(* CODESYS project SPT_Components.library
   Company: Beckhoff Automation LLC
   DefaultNamespace: SPT_Components
   Version: 3.9.2
   Placeholder: SPT Components
   Title: SPT Components

Project tree, tasks and I/O mapping:
  libraries: SPT Base Types, * (Beckhoff Automation LLC); SPT Event Logger, * (Beckhoff Automation LLC); SPT Motion Control, * (Beckhoff Automation LLC); SPT Utilities, * (Beckhoff Automation LLC); Tc2_DataExchange, * (Beckhoff Automation GmbH); Tc2_EtherCAT, * (Beckhoff Automation GmbH); Tc2_MC2, * (Beckhoff Automation GmbH); Tc2_ModbusRTU, * (Beckhoff Automation GmbH); Tc2_Standard, * (Beckhoff Automation GmbH); Tc2_System, * (Beckhoff Automation GmbH); Tc2_Utilities, * (Beckhoff Automation GmbH); Tc3_EventLogger, * (Beckhoff Automation GmbH); Tc3_Module, * (Beckhoff Automation GmbH); Tc3_PackML_V2, * (Beckhoff Automation GmbH)
  Axes/
    DUT/
      data type ST_AxisBase_Command
      data type ST_AxisBase_Config
      data type ST_AxisBase_HMI
      data type ST_AxisBase_Status
    function block FB_Component_BasicAxis [ST]: Disable, Enable, Home, Jog, MoveAbsolute, MoveModulo, MoveRelative, MoveVelocity, ReadParameterSet, Reset, RunExternalSequence, Stop, WriteBoolParameter, WriteParameter, Acceleration, Deceleration, Jerk, Velocity, ActualAcceleration, ActualPosition, ActualPositionModulo, ActualTorque, ActualVelocity, PositionLag, SetAcceleration, SetPosition, SetPositionModulo, SetVelocity, Enabled, InPosition, Stopped, Axis, AxisParameters, ExternalSequence, HomeMethod, InhibitFeedNegative, InhibitFeedPositive, Override, ResetMethod, CreateEvents, HMICommunication, Monitoring, CyclicLogic, Initialize
    function block FB_Component_BasicSlaveAxis [ST]: Disable, Enable, Home, Jog, MoveAbsolute, MoveModulo, MoveRelative, MoveVelocity, ReadParameterSet, Reset, RunExternalSequence, Stop, WriteBoolParameter, WriteParameter, Acceleration, Deceleration, Jerk, Velocity, ActualAcceleration, ActualPosition, ActualPositionModulo, ActualTorque, ActualVelocity, PositionLag, SetAcceleration, SetPosition, SetPositionModulo, SetVelocity, Enabled, InPosition, Stopped, Axis, AxisParameters, ExternalSequence, HomeMethod, InhibitFeedNegative, InhibitFeedPositive, Override, ResetMethod, GearIn, GearOut, InGear, Master1, Master2, Master3, Master4, RatioMaster1, RatioMaster2, RatioMaster3, RatioMaster4, CreateEvents, HMICommunication, Monitoring, CyclicLogic, Initialize
    function block FB_Component_CamSlaveAxis [ST]: Disable, Enable, Home, Jog, MoveAbsolute, MoveModulo, MoveRelative, MoveVelocity, ReadParameterSet, Reset, RunExternalSequence, Stop, WriteBoolParameter, WriteParameter, Acceleration, Deceleration, Jerk, Velocity, ActualAcceleration, ActualPosition, ActualPositionModulo, ActualTorque, ActualVelocity, PositionLag, SetAcceleration, SetPosition, SetPositionModulo, SetVelocity, Enabled, InPosition, Stopped, Axis, AxisParameters, ExternalSequence, HomeMethod, InhibitFeedNegative, InhibitFeedPositive, Override, ResetMethod, CamParameters, ChangeMode, FindSlavePos, FindSyncPos, InSync, Master, RunningTable, StartCouple, StartSync, SyncPos, UpdateTable, WaitingForCommand, CreateEvents, HMICommunication, Monitoring, CyclicLogic, Initialize
  Communications/
    Modbus-RTU/
      function block FB_Component_ModbusRTUMaster [ST]: CreateEvents, CyclicLogic, Initialize, Monitoring, Reset, RegisterAsyncRequest, RegisterSyncRequest, ProcessRead, ProcessWrite
      function block FB_ModbusAsyncQueue [ST]: Clear, Count, Dequeue, Enqueue, NextRequest
      function block FB_ModbusSyncQueue [ST]: Clear, Count, Enqueue, NextRequest
      interface I_ModbusConsumer: ModbusRequestComplete, SlaveID
      interface I_ModbusProvider: RegisterAsyncRequest, RegisterSyncRequest
      global variables Parameters_ModbusRTU
      data type ST_ModbusOperation
      data type ST_ModbusRequest
  GVLs/
    global variables CONSTANTS
  PackML/
    DUT/
      data type ST_EventInfo
      data type ST_PackML_aEventInfo
      data type ST_PackML_aMsgState
    function block FB_Component_PackML_EventHandler [ST]: AdminTag, AlarmArrayHandler, AlarmToStopReason, AllowHMIControl, BlockHMIControl, Busy, ClearStopReason, ConfirmAlarm, CurrentAlarmSeverity, CyclicLogic, Error, ErrorID, EventListener, Execute, GetMsgInfos, InitComplete, Initialize, InSimulation, InternalErrorAck, MoveAlarmToHistory, Name, OnAlarmCleared, OnAlarmConfirmed, OnAlarmRaised, ParentResponseDefinitions, Reset, TimeZone, WarningToStopReason, WriteAlarmTags
  Project Information/
    function F_GetCompany [ST]
    function F_GetTitle [ST]
    function F_GetVersion [ST]
  Sensors/
    DUT/
      data type E_DebounceMode
      data type E_SensorSimulationMode
      data type ST_DigitalSensor_Command
      data type ST_DigitalSensor_Config
      data type ST_DigitalSensor_HMI
      data type ST_DigitalSensor_Status
    function block FB_DigitalSensor [ST]: CyclicLogic, Active, DebounceMode, DebounceTime, Inverted, SimulationInput, SimulationMode, SimulationTimeBase, TimeActive, TimeInactive, HMICommunication, Monitoring, ProcessInput
    interface I_DigitalSensorBase: Active, DebounceMode, DebounceTime, Inverted, SimulationInput, SimulationMode, TimeActive, TimeInactive
  Solenoids/
    DUT/
      data type ST_Cylinder_Command
      data type ST_Cylinder_Config
      data type ST_Cylinder_HMI
      data type ST_Cylinder_Status
    SolenoidBankBase/
      data type E_SolenoidType
      function block FB_SolenoidBankBase [ST]: AddSolenoid, CheckNumber, CreateEvents, CyclicLogic, Initialize, MapIO, Monitoring, Reset
      data type ST_SolenoidBankConfig
    function block FB_DoubleSolenoid [ST]: HardwareInit, HardwareUpdate, RetractOutput
    function block FB_DoubleSolenoidFeedback [ST]: ExtendedInput, Feedback, HardwareInit, RetractedInput
    function block FB_SingleSolenoid [ST]: CreateEvents, HMICommunication, Monitoring, CyclicLogic, Extend, Extended, ExtendOutput, ExtendTime, Retract, Retracted, RetractOutput, RetractTime, Feedback, HardwareInit, HardwareUpdate, Initialize, Reset
    function block FB_SingleSolenoidFeedback [ST]: ExtendedInput, Feedback, HardwareInit, RetractedInput
    interface I_Solenoid: Extend, Extended, ExtendOutput, ExtendTime, Retract, Retracted, RetractOutput, RetractTime
    global variables Parameters_Cylinder
  Version/
    global variables Global_Version
  00000000-0000-0000-0000-000000000000|LICENSE
  LICENSE
*)

// Axes/DUT/ST_AxisBase_Command
{attribute 'OPC.UA.DA' := '1'}
{attribute 'OPC.UA.DA.StructuredType' := '1'}
{attribute 'OPC.UA.DA.Access' := '3'}
TYPE ST_AxisBase_Command :
	STRUCT
		JogFast_Forward	 : BOOL;
		JogFast_Backward : BOOL;
		JogSlow_Forward	 : BOOL;
		JogSlow_Backward : BOOL;
	END_STRUCT
END_TYPE

// Axes/DUT/ST_AxisBase_Config
{attribute 'OPC.UA.DA' := '1'}
{attribute 'OPC.UA.DA.StructuredType' := '1'}
{attribute 'OPC.UA.DA.Access' := '1'}
TYPE ST_AxisBase_Config :
	STRUCT
	END_STRUCT
END_TYPE

// Axes/DUT/ST_AxisBase_HMI
{attribute 'OPC.UA.DA' := '1'}
{attribute 'OPC.UA.DA.StructuredType' := '1'}
TYPE ST_AxisBase_HMI :
	STRUCT
		Config	: ST_AxisBase_Config;
		Command : ST_AxisBase_Command;
		Status	: ST_AxisBase_Status;
	END_STRUCT
END_TYPE

// Axes/DUT/ST_AxisBase_Status
{attribute 'OPC.UA.DA' := '1'}
{attribute 'OPC.UA.DA.StructuredType' := '1'}
{attribute 'OPC.UA.DA.Access' := '1'}
TYPE ST_AxisBase_Status :
	STRUCT
		Enabled				 : BOOL;
		InPosition			 : BOOL;
		Stopped				 : BOOL;
		Coupled				 : BOOL;
		SetPosition			 : LREAL;
		SetPositionModulo	 : LREAL;
		SetVelocity			 : LREAL;
		SetAcceleration		 : LREAL;
		ActualPosition		 : LREAL;
		ActualPositionModulo : LREAL;
		ActualVelocity		 : LREAL;
		ActualAcceleration	 : LREAL;
		ActualTorque		 : LREAL;
		PositionLag			 : LREAL;
	END_STRUCT
END_TYPE

// Communications/Modbus-RTU/ST_ModbusOperation
TYPE ST_ModbusOperation :
	STRUCT
		StartAddress : UINT;
		EndAddress	 : UINT;
		pAddress	 : PVOID;
	END_STRUCT
END_TYPE

// Communications/Modbus-RTU/ST_ModbusRequest
TYPE ST_ModbusRequest :
	STRUCT
		ipRequestor : I_ModbusConsumer;
		RequestID	: ULINT;
		ReadOps		: ARRAY[1..Parameters_ModbusRTU.MAX_MODBUS_RW_OPS_PER_REQUEST] OF ST_ModbusOperation;
		WriteOps	: ARRAY[1..Parameters_ModbusRTU.MAX_MODBUS_RW_OPS_PER_REQUEST] OF ST_ModbusOperation;
	END_STRUCT
END_TYPE

// PackML/DUT/ST_EventInfo
TYPE ST_EventInfo :
	STRUCT
		eSeverity		   : TCEVENTSEVERITY;
		EventClass		   : GUID;
		EventId			   : UDINT;
		ipArguments		   : I_TcArguments;
		fbRequestEventText : FB_RequestEventText;
		EventText		   : STRING;
		Source			   : STRING;
		TimeRaised		   : ARRAY[0..6] OF DINT;
		TimeConfirmed	   : ARRAY[0..6] OF DINT;
		TimeCleared		   : ARRAY[0..6] OF DINT;
	END_STRUCT
END_TYPE

// PackML/DUT/ST_PackML_aEventInfo
TYPE ST_PackML_aEventInfo :
	STRUCT
		Warning		  : ST_PackML_aMsgState; // Warning Informatins
		Alarm		  : ST_PackML_aMsgState; // Alarm Informations
		StopReason	  : ST_PackML_aMsgState; // StopReason Informations
		HistorizedMsg : UDINT;				 // Number of historized Messages
	END_STRUCT
END_TYPE

// PackML/DUT/ST_PackML_aMsgState
TYPE ST_PackML_aMsgState :
	STRUCT
		Active			: BOOL;	 // a unconfirmed Message is pending
		NumberActive	: UDINT; // Number of active Messages
		NumberConfirmed : UDINT; // Number of confirmed Messages			
		NumberCleared	: UDINT; // Number of Cleared Messages in History
	END_STRUCT
END_TYPE

// Sensors/DUT/E_DebounceMode
{attribute 'qualified_only'}
{attribute 'strict'}
TYPE E_DebounceMode : (
		RawInput,
		SimpleFlickerFilter,
		EdgeDetectFilter,
		MovingAverage
	) DINT;
END_TYPE

// Sensors/DUT/E_SensorSimulationMode
{attribute 'qualified_only'}
{attribute 'strict'}
TYPE E_SensorSimulationMode : (
		InputDriven, // Follows the state of the SimulationInput property
		Periodic	 // Follows a 50% duty cycle at the period specified in ms by SimulationInput);
	);
END_TYPE

// Sensors/DUT/ST_DigitalSensor_Command
{attribute 'OPC.UA.DA' := '1'}
{attribute 'OPC.UA.DA.StructuredType' := '1'}
{attribute 'OPC.UA.DA.Access' := '3'}
TYPE ST_DigitalSensor_Command :
	STRUCT
	END_STRUCT
END_TYPE

// Sensors/DUT/ST_DigitalSensor_Config
{attribute 'OPC.UA.DA' := '1'}
{attribute 'OPC.UA.DA.StructuredType' := '1'}
{attribute 'OPC.UA.DA.Access' := '1'}
TYPE ST_DigitalSensor_Config :
	STRUCT
		// Status information
		DebounceMode	   : E_DebounceMode;
		DebounceTime	   : TIME;
		Inverted		   : BOOL;
		SimulationMode	   : E_SensorSimulationMode;
		SimulationTimebase : UDINT;
	END_STRUCT
END_TYPE

// Sensors/DUT/ST_DigitalSensor_HMI
{attribute 'OPC.UA.DA' := '1'}
{attribute 'OPC.UA.DA.StructuredType' := '1'}
TYPE ST_DigitalSensor_HMI :
	STRUCT
		Config	: ST_DigitalSensor_Config;
		Command : ST_DigitalSensor_Command;
		Status	: ST_DigitalSensor_Status;
	END_STRUCT
END_TYPE

// Sensors/DUT/ST_DigitalSensor_Status
{attribute 'OPC.UA.DA' := '1'}
{attribute 'OPC.UA.DA.StructuredType' := '1'}
{attribute 'OPC.UA.DA.Access' := '1'}
TYPE ST_DigitalSensor_Status :
	STRUCT
		Active		 : BOOL;
		TimeActive	 : LREAL;
		TimeInactive : LREAL;
	END_STRUCT
END_TYPE

// Solenoids/DUT/ST_Cylinder_Command
{attribute 'OPC.UA.DA' := '1'}
{attribute 'OPC.UA.DA.StructuredType' := '1'}
{attribute 'OPC.UA.DA.Access' := '3'}
TYPE ST_Cylinder_Command :
	STRUCT
		Extend		: BOOL;
		Retract		: BOOL;
		ExtendTime	: LREAL;
		RetractTime : LREAL;
	END_STRUCT
END_TYPE

// Solenoids/DUT/ST_Cylinder_Config
{attribute 'OPC.UA.DA' := '1'}
{attribute 'OPC.UA.DA.StructuredType' := '1'}
{attribute 'OPC.UA.DA.Access' := '1'}
TYPE ST_Cylinder_Config :
	STRUCT
		ExtendTime	: LREAL;
		RetractTime : LREAL;
	END_STRUCT
END_TYPE

// Solenoids/DUT/ST_Cylinder_HMI
{attribute 'OPC.UA.DA' := '1'}
{attribute 'OPC.UA.DA.StructuredType' := '1'}
TYPE ST_Cylinder_HMI :
	STRUCT
		Config	: ST_Cylinder_Config;
		Command : ST_Cylinder_Command;
		Status	: ST_Cylinder_Status;
	END_STRUCT
END_TYPE

// Solenoids/DUT/ST_Cylinder_Status
{attribute 'OPC.UA.DA' := '1'}
{attribute 'OPC.UA.DA.StructuredType' := '1'}
{attribute 'OPC.UA.DA.Access' := '1'}
TYPE ST_Cylinder_Status :
	STRUCT
		Extended   : BOOL;
		Retracted  : BOOL;
		Extending  : BOOL;
		Retracting : BOOL;
	END_STRUCT
END_TYPE

// Solenoids/SolenoidBankBase/E_SolenoidType
{attribute 'qualified_only'}
{attribute 'strict'}
TYPE E_SolenoidType : (
		Single,
		Double,
		SingleFeedback,
		DoubleFeedback
	);
END_TYPE

// Solenoids/SolenoidBankBase/ST_SolenoidBankConfig
TYPE ST_SolenoidBankConfig :
	STRUCT
		SolenoidType		 : E_SolenoidType;
		ipSolenoid			 : I_Solenoid;
		SolenoidOutputNumber : UINT;
	END_STRUCT
END_TYPE

// Communications/Modbus-RTU/Parameters_ModbusRTU
{attribute 'qualified_only'}
VAR_GLOBAL CONSTANT
	MAX_MODBUS_REQUESTS			  : UDINT := 100;
	MAX_MODBUS_RW_OPS_PER_REQUEST : UDINT := 100;
	MODBUS_TIMEOUT				  : TIME  := T#100MS;
END_VAR

// GVLs/CONSTANTS
{attribute 'qualified_only'}
VAR_GLOBAL CONSTANT
	BASIC_AXIS_ALARM_COUNT		 : UINT := 18;
	BASIC_SLAVE_AXIS_ALARM_COUNT : UINT := 3;
	CAM_SLAVE_AXIS_ALARM_COUNT	 : UINT := 9;
END_VAR

// Solenoids/Parameters_Cylinder
{attribute 'qualified_only'}
VAR_GLOBAL CONSTANT
	MAX_NUMBER_OF_SOLENOIDS : UINT := 32;
END_VAR

// Version/Global_Version
{attribute 'TcGenerated'}
{attribute 'no-analysis'}
{attribute 'linkalways'}

// This function has been automatically generated from the project information.
VAR_GLOBAL CONSTANT
	{attribute 'const_non_replaced'}
	stLibVersion_SPT_Components : ST_LibVersion := (iMajor := 3, iMinor := 9, iBuild := 2, iRevision := 0, nFlags := 1, sVersion := '3.9.2');
END_VAR

// Axes/FB_Component_BasicAxis
FUNCTION_BLOCK FB_Component_BasicAxis EXTENDS FB_ComponentBase IMPLEMENTS I_BasicAxis
VAR
	BasicAxis						  : FB_BasicAxis;
	AxisBase_HMI					  : ST_AxisBase_HMI;
	BasicAxisAlarms					  : ARRAY[1..CONSTANTS.BASIC_AXIS_ALARM_COUNT] OF FB_TcAlarm;
	HMICommand_BasicAxis_RT			  : R_TRIG;
	ResetPreviouslyErrored			  : BOOL;
	HomePreviouslyErrored			  : BOOL;
	ExternalSequencePreviouslyErrored : BOOL;
END_VAR

// There should be no code in the function block body of a class that Implements I_CyclicFB

METHOD Disable : BOOL
Disable := BasicAxis.Disable();
END_METHOD

METHOD Enable : BOOL
Enable := BasicAxis.Enable();
END_METHOD

METHOD Home : BOOL
IF BasicAxis.Home() THEN
	HomePreviouslyErrored := FALSE;
	Home				  := TRUE;
END_IF
END_METHOD

METHOD Jog : BOOL
VAR_INPUT
	JogFW	 : BOOL;
	JogBW	 : BOOL;
	JogMode	 : E_JogMode;
	Position : LREAL;
END_VAR
Jog := BasicAxis.Jog(JogFW,
					 JogBW,
					 JogMode,
					 Position);
END_METHOD

METHOD MoveAbsolute : BOOL
VAR_INPUT
	Position	  : LREAL;
	AbortPrevious : BOOL;
END_VAR
MoveAbsolute := BasicAxis.MoveAbsolute(Position, AbortPrevious);
END_METHOD

METHOD MoveModulo : BOOL
VAR_INPUT
	Position	  : LREAL;
	Direction	  : MC_Direction;
	AbortPrevious : BOOL;
END_VAR
MoveModulo := BasicAxis.MoveModulo(Position, Direction, AbortPrevious);
END_METHOD

METHOD MoveRelative : BOOL
VAR_INPUT
	Distance	  : LREAL;
	AbortPrevious : BOOL;
END_VAR
MoveRelative := BasicAxis.MoveRelative(Distance, AbortPrevious);
END_METHOD

METHOD MoveVelocity : BOOL
VAR_INPUT
	Velocity	  : LREAL;
	AbortPrevious : BOOL;
END_VAR
MoveVelocity := BasicAxis.MoveVelocity(Velocity, AbortPrevious);
END_METHOD

METHOD ReadParameterSet : BOOL
VAR_INPUT
END_VAR
ReadParameterSet := BasicAxis.ReadParameterSet();
END_METHOD

METHOD Reset : BOOL
Reset := FALSE;
SUPER^.Reset();
IF BasicAxis.ResetMethod <> 0 THEN
	IF (BasicAxis.ResetMethod.Error AND ResetPreviouslyErrored) AND BasicAxisAlarms[E_BasicAxis.ResetError].bRaised THEN
		BasicAxisAlarms[E_BasicAxis.ResetError].Clear(0, 0);
	END_IF
END_IF

IF BasicAxis.HomeMethod <> 0 THEN
	IF (BasicAxis.HomeMethod.Error AND HomePreviouslyErrored) AND BasicAxisAlarms[E_BasicAxis.HomeError].bRaised THEN
		BasicAxisAlarms[E_BasicAxis.HomeError].Clear(0, 0);
	END_IF
END_IF

IF BasicAxis.ExternalSequence <> 0 THEN
	IF (BasicAxis.ExternalSequence.Error AND ExternalSequencePreviouslyErrored) AND BasicAxisAlarms[E_BasicAxis.ExternalSequenceError].bRaised THEN
		BasicAxisAlarms[E_BasicAxis.ExternalSequenceError].Clear(0, 0);
	END_IF
END_IF

IF BasicAxis.Reset() THEN
	_Error				   := FALSE;
	_ErrorID			   := 0;
	ResetPreviouslyErrored := FALSE;
	Reset				   := TRUE;
END_IF
END_METHOD

METHOD RunExternalSequence : BOOL
IF BasicAxis.RunExternalSequence() THEN
	ExternalSequencePreviouslyErrored := FALSE;
	RunExternalSequence				  := TRUE;
END_IF
END_METHOD

METHOD Stop : BOOL
Stop := BasicAxis.Stop();
END_METHOD

METHOD WriteBoolParameter : BOOL
VAR_INPUT
	ParameterNumber : MC_AxisParameter;
	Value			: BOOL;
END_VAR
WriteBoolParameter := BasicAxis.WriteBoolParameter(ParameterNumber, Value);
END_METHOD

METHOD WriteParameter : BOOL
VAR_INPUT
	ParameterNumber : MC_AxisParameter;
	Value			: LREAL;
END_VAR
WriteParameter := BasicAxis.WriteParameter(ParameterNumber, Value);
END_METHOD

PROPERTY Acceleration : LREAL
GET
Acceleration := BasicAxis.Acceleration;
END_GET
SET
BasicAxis.Acceleration := Acceleration;
END_SET
END_PROPERTY

PROPERTY Deceleration : LREAL
GET
Deceleration := BasicAxis.Deceleration;
END_GET
SET
BasicAxis.Deceleration := Deceleration;
END_SET
END_PROPERTY

PROPERTY Jerk : LREAL
GET
Jerk := BasicAxis.Jerk;
END_GET
SET
BasicAxis.Jerk := Jerk;
END_SET
END_PROPERTY

PROPERTY Velocity : LREAL
GET
Velocity := BasicAxis.Velocity;
END_GET
SET
BasicAxis.Velocity := Velocity;
END_SET
END_PROPERTY

PROPERTY ActualAcceleration : LREAL
GET
ActualAcceleration := BasicAxis.ActualAcceleration;
END_GET
END_PROPERTY

PROPERTY ActualPosition : LREAL
GET
ActualPosition := BasicAxis.ActualPosition;
END_GET
END_PROPERTY

PROPERTY ActualPositionModulo : LREAL
GET
ActualPositionModulo := BasicAxis.ActualPositionModulo;
END_GET
END_PROPERTY

PROPERTY ActualTorque : LREAL
GET
ActualTorque := BasicAxis.ActualTorque;
END_GET
END_PROPERTY

PROPERTY ActualVelocity : LREAL
GET
ActualVelocity := BasicAxis.ActualVelocity;
END_GET
END_PROPERTY

PROPERTY PositionLag : LREAL
GET
PositionLag := BasicAxis.PositionLag;
END_GET
END_PROPERTY

PROPERTY SetAcceleration : LREAL
GET
SetAcceleration := BasicAxis.SetAcceleration;
END_GET
END_PROPERTY

PROPERTY SetPosition : LREAL
GET
SetPosition := BasicAxis.SetPosition;
END_GET
END_PROPERTY

PROPERTY SetPositionModulo : LREAL
GET
SetPositionModulo := BasicAxis.SetPositionModulo;
END_GET
END_PROPERTY

PROPERTY SetVelocity : LREAL
GET
SetVelocity := BasicAxis.SetVelocity;
END_GET
END_PROPERTY

PROPERTY Enabled : BOOL
GET
Enabled := BasicAxis.Enabled;
END_GET
END_PROPERTY

PROPERTY InPosition : BOOL
GET
InPosition := BasicAxis.InPosition;
END_GET
END_PROPERTY

PROPERTY Stopped : BOOL
GET
Stopped := BasicAxis.Stopped;
END_GET
END_PROPERTY

{attribute 'analysis' := '-29'}
PROPERTY Axis : REFERENCE TO AXIS_REF
GET
Axis REF= BasicAxis.Axis;
END_GET
END_PROPERTY

PROPERTY AxisParameters : REFERENCE TO ST_AxisParameterSet
GET
AxisParameters REF= BasicAxis.AxisParameters;
END_GET
END_PROPERTY

PROPERTY ExternalSequence : I_MotionSequence
GET
ExternalSequence := BasicAxis.ExternalSequence;
END_GET
SET
BasicAxis.ExternalSequence := ExternalSequence;
END_SET
END_PROPERTY

PROPERTY HomeMethod : I_MotionSequence
SET
BasicAxis.HomeMethod := HomeMethod;
END_SET
END_PROPERTY

PROPERTY InhibitFeedNegative : BOOL
GET
InhibitFeedNegative := BasicAxis.InhibitFeedNegative;
END_GET
SET
BasicAxis.InhibitFeedNegative := InhibitFeedNegative;
END_SET
END_PROPERTY

PROPERTY InhibitFeedPositive : BOOL
GET
InhibitFeedPositive := BasicAxis.InhibitFeedPositive;
END_GET
SET
BasicAxis.InhibitFeedPositive := InhibitFeedPositive;
END_SET
END_PROPERTY

PROPERTY Override : LREAL
GET
Override := BasicAxis.Override;
END_GET
SET
IF Override >= 0 AND Override <= 100 THEN
	BasicAxis.Override := Override;
END_IF
END_SET
END_PROPERTY

PROPERTY ResetMethod : I_MotionSequence
GET
ResetMethod := BasicAxis.ResetMethod;
END_GET
SET
BasicAxis.ResetMethod := ResetMethod;
END_SET
END_PROPERTY

METHOD PROTECTED CreateEvents
F_CreateAllEventsInClass(Alarms		:= BasicAxisAlarms,
						 ClassSize	:= SIZEOF(TC_EVENTS.BasicAxis),
						 pInitEvent := ADR(TC_EVENTS.BasicAxis.InitReferenceEvent),
						 Prefix		:= Name);

SUPER^.CreateEvents();
END_METHOD

METHOD PROTECTED HMICommunication
// Extend this method in extended FBs to communicate specific implementation data
SUPER^.HMICommunication();

// Process HMI requests

// Replace 'FALSE' below with further momentary commands (myCommand XOR myOtherCommand XOR...)
HMICommand_BasicAxis_RT(CLK := (ComponentBase_HMI.Status.HMIControlAvailable AND NOT HMICommandActive_Base));

// Signal to FB_ComponentBase that a command is active
HMICommandActive_Descendant := ComponentBase_HMI.Status.HMIControlAvailable AND (AxisBase_HMI.Command.JogFast_Backward OR AxisBase_HMI.Command.JogFast_Forward OR AxisBase_HMI.Command.JogSlow_Forward OR AxisBase_HMI.Command.JogSlow_Backward);

// Process HMI requests
IF HMICommand_BasicAxis_RT.Q THEN // If a request has been issued by the HMI, and a previous request has not just finished being processed
END_IF

IF ComponentBase_HMI.Status.HMIControlAvailable AND NOT HMICommand_BasicAxis_RT.Q THEN
	IF AxisBase_HMI.Command.JogSlow_Forward THEN
		BasicAxis.Jog(AxisBase_HMI.Command.JogSlow_Forward,
					  FALSE,
					  E_JogMode.MC_JOGMODE_STANDARD_SLOW,
					  0.0);
	ELSIF AxisBase_HMI.Command.JogSlow_Backward THEN
		BasicAxis.Jog(FALSE,
					  AxisBase_HMI.Command.JogSlow_Backward,
					  E_JogMode.MC_JOGMODE_STANDARD_SLOW,
					  0.0);
	ELSIF AxisBase_HMI.Command.JogFast_Forward THEN
		BasicAxis.Jog(AxisBase_HMI.Command.JogFast_Forward,
					  FALSE,
					  E_JogMode.MC_JOGMODE_STANDARD_FAST,
					  0.0);
	ELSIF AxisBase_HMI.Command.JogFast_Backward THEN
		BasicAxis.Jog(FALSE,
					  AxisBase_HMI.Command.JogFast_Backward,
					  E_JogMode.MC_JOGMODE_STANDARD_FAST,
					  0.0);
	ELSE
		BasicAxis.Jog(FALSE,
					  FALSE,
					  E_JogMode.MC_JOGMODE_STANDARD_SLOW,
					  0.0);
	END_IF
END_IF

// Update HMI status info
AxisBase_HMI.Status.Enabled				 := BasicAxis.Enabled;
AxisBase_HMI.Status.InPosition			 := BasicAxis.InPosition;
AxisBase_HMI.Status.Stopped				 := BasicAxis.Stopped;
AxisBase_HMI.Status.Coupled				 := FALSE;
AxisBase_HMI.Status.SetPosition			 := BasicAxis.SetPosition;
AxisBase_HMI.Status.SetPositionModulo	 := BasicAxis.SetPositionModulo;
AxisBase_HMI.Status.SetVelocity			 := BasicAxis.SetVelocity;
AxisBase_HMI.Status.SetAcceleration		 := BasicAxis.SetAcceleration;
AxisBase_HMI.Status.ActualPosition		 := BasicAxis.ActualPosition;
AxisBase_HMI.Status.ActualPositionModulo := BasicAxis.ActualPositionModulo;
AxisBase_HMI.Status.ActualVelocity		 := BasicAxis.ActualVelocity;
AxisBase_HMI.Status.ActualAcceleration	 := BasicAxis.ActualAcceleration;
AxisBase_HMI.Status.ActualTorque		 := BasicAxis.ActualTorque;
AxisBase_HMI.Status.PositionLag			 := BasicAxis.PositionLag;
END_METHOD

METHOD PROTECTED Monitoring
SUPER^.Monitoring();

// ErrorID 2 - MC_Power
IF BasicAxis.MCPower.Error AND NOT BasicAxisAlarms[E_BasicAxis.PowerError].bRaised THEN
	RaiseAlarmWithStrings(Alarm := BasicAxisAlarms[E_BasicAxis.PowerError], UDINT_TO_STRING(BasicAxis.ErrorID), '');
ELSIF NOT BasicAxis.MCPower.Error AND BasicAxisAlarms[E_BasicAxis.PowerError].bRaised THEN
	BasicAxisAlarms[E_BasicAxis.PowerError].Clear(0, 0);
END_IF

// ErrorID 3 - MC_Reset (or other reset method)
IF BasicAxis.ResetMethod <> 0 THEN
	IF (BasicAxis.ResetMethod.Error AND NOT ResetPreviouslyErrored) AND NOT BasicAxisAlarms[E_BasicAxis.ResetError].bRaised THEN
		ResetPreviouslyErrored := TRUE;
		RaiseAlarmWithStrings(Alarm := BasicAxisAlarms[E_BasicAxis.ResetError], UDINT_TO_STRING(BasicAxis.ResetMethod.ErrorID), '');
	ELSIF NOT BasicAxis.ResetMethod.Error AND BasicAxisAlarms[E_BasicAxis.ResetError].bRaised THEN
		BasicAxisAlarms[E_BasicAxis.ResetError].Clear(0, 0);
	END_IF
END_IF

// ErrorID 4 - MC_Halt
IF BasicAxis.MCHalt.Error AND NOT BasicAxisAlarms[E_BasicAxis.HaltError].bRaised THEN
	RaiseAlarmWithStrings(Alarm := BasicAxisAlarms[E_BasicAxis.HaltError], UDINT_TO_STRING(BasicAxis.MCHalt.ErrorID), '');
ELSIF NOT BasicAxis.MCHalt.Error AND BasicAxisAlarms[E_BasicAxis.HaltError].bRaised THEN
	BasicAxisAlarms[E_BasicAxis.HaltError].Clear(0, 0);
END_IF

// ErrorID 5 - MC_Stop **NOT IMPLEMENTED**

// ErrorID 6 - MC_Home (or other home method)
IF BasicAxis.HomeMethod <> 0 THEN
	IF (BasicAxis.HomeMethod.Error AND NOT HomePreviouslyErrored) AND NOT BasicAxisAlarms[E_BasicAxis.HomeError].bRaised THEN
		HomePreviouslyErrored := TRUE;
		RaiseAlarmWithStrings(Alarm := BasicAxisAlarms[E_BasicAxis.HomeError], UDINT_TO_STRING(BasicAxis.HomeMethod.ErrorID), '');
	ELSIF NOT BasicAxis.HomeMethod.Error AND BasicAxisAlarms[E_BasicAxis.HomeError].bRaised THEN
		BasicAxisAlarms[E_BasicAxis.HomeError].Clear(0, 0);
	END_IF
END_IF

// ErrorID 7 - MC_Jog 
IF BasicAxis.MCJog.Error AND NOT BasicAxisAlarms[E_BasicAxis.JogError].bRaised THEN
	RaiseAlarmWithStrings(Alarm := BasicAxisAlarms[E_BasicAxis.JogError], UDINT_TO_STRING(BasicAxis.MCJog.ErrorID), '');
ELSIF NOT BasicAxis.MCJog.Error AND BasicAxisAlarms[E_BasicAxis.JogError].bRaised THEN
	BasicAxisAlarms[E_BasicAxis.JogError].Clear(0, 0);
END_IF

// ErrorID 8 - MC_MoveAbsolute
IF BasicAxis.MCMoveAbsolute <> 0 THEN
	IF BasicAxis.MCMoveAbsolute^.Error AND NOT BasicAxisAlarms[E_BasicAxis.MoveAbsoluteError].bRaised THEN
		RaiseAlarmWithStrings(Alarm := BasicAxisAlarms[E_BasicAxis.MoveAbsoluteError], UDINT_TO_STRING(BasicAxis.MCMoveAbsolute^.ErrorID), '');
	ELSIF NOT BasicAxis.MCMoveAbsolute^.Error AND BasicAxisAlarms[E_BasicAxis.MoveAbsoluteError].bRaised THEN
		BasicAxisAlarms[E_BasicAxis.MoveAbsoluteError].Clear(0, 0);
	END_IF
END_IF

// ErrorID 9 - MC_MoveRelative
IF BasicAxis.MCMoveRelative <> 0 THEN
	IF BasicAxis.MCMoveRelative^.Error AND NOT BasicAxisAlarms[E_BasicAxis.MoveRelativeError].bRaised THEN
		RaiseAlarmWithStrings(Alarm := BasicAxisAlarms[E_BasicAxis.MoveRelativeError], UDINT_TO_STRING(BasicAxis.MCMoveRelative^.ErrorID), '');
	ELSIF NOT BasicAxis.MCMoveRelative^.Error AND BasicAxisAlarms[E_BasicAxis.MoveRelativeError].bRaised THEN
		BasicAxisAlarms[E_BasicAxis.MoveRelativeError].Clear(0, 0);
	END_IF
END_IF

// ErrorID 10 - MC_MoveVelocity
IF BasicAxis.MCMoveVelocity <> 0 THEN
	IF BasicAxis.MCMoveVelocity^.Error AND NOT BasicAxisAlarms[E_BasicAxis.MoveVelocityError].bRaised THEN
		RaiseAlarmWithStrings(Alarm := BasicAxisAlarms[E_BasicAxis.MoveVelocityError], UDINT_TO_STRING(BasicAxis.MCMoveVelocity^.ErrorID), '');
	ELSIF NOT BasicAxis.MCMoveVelocity^.Error AND BasicAxisAlarms[E_BasicAxis.MoveVelocityError].bRaised THEN
		BasicAxisAlarms[E_BasicAxis.MoveVelocityError].Clear(0, 0);
	END_IF
END_IF

// ErrorID 11 - MC_MoveModulo
IF BasicAxis.MCMoveModulo <> 0 THEN
	IF BasicAxis.MCMoveModulo^.Error AND NOT BasicAxisAlarms[E_BasicAxis.MoveModuloError].bRaised THEN
		RaiseAlarmWithStrings(Alarm := BasicAxisAlarms[E_BasicAxis.MoveModuloError], UDINT_TO_STRING(BasicAxis.MCMoveModulo^.ErrorID), '');
	ELSIF NOT BasicAxis.MCMoveModulo^.Error AND BasicAxisAlarms[E_BasicAxis.MoveModuloError].bRaised THEN
		BasicAxisAlarms[E_BasicAxis.MoveModuloError].Clear(0, 0);
	END_IF
END_IF

// ErrorID 12 - MC_ReadParameterSet
IF BasicAxis.MCReadParameterSet.Error AND NOT BasicAxisAlarms[E_BasicAxis.ReadParameterSetError].bRaised THEN
	RaiseAlarmWithStrings(Alarm := BasicAxisAlarms[E_BasicAxis.ReadParameterSetError], UDINT_TO_STRING(BasicAxis.MCReadParameterSet.ErrorID), '');
ELSIF NOT BasicAxis.MCReadParameterSet.Error AND BasicAxisAlarms[E_BasicAxis.ReadParameterSetError].bRaised THEN
	BasicAxisAlarms[E_BasicAxis.ReadParameterSetError].Clear(0, 0);
END_IF

// ErrorID 13 - MC_WriteParameter
IF BasicAxis.MCWriteParameter.Error AND NOT BasicAxisAlarms[E_BasicAxis.WriteParameterError].bRaised THEN
	RaiseAlarmWithStrings(Alarm := BasicAxisAlarms[E_BasicAxis.WriteParameterError], UDINT_TO_STRING(BasicAxis.MCWriteParameter.ErrorID), '');
ELSIF NOT BasicAxis.MCWriteParameter.Error AND BasicAxisAlarms[E_BasicAxis.WriteParameterError].bRaised THEN
	BasicAxisAlarms[E_BasicAxis.WriteParameterError].Clear(0, 0);
END_IF

// ErrorID 14 - MC_WriteBoolParameter
IF BasicAxis.MCWriteBoolParameter.Error AND NOT BasicAxisAlarms[E_BasicAxis.WriteBoolParameterError].bRaised THEN
	RaiseAlarmWithStrings(Alarm := BasicAxisAlarms[E_BasicAxis.WriteBoolParameterError], UDINT_TO_STRING(BasicAxis.MCWriteBoolParameter.ErrorID), '');
ELSIF NOT BasicAxis.MCWriteBoolParameter.Error AND BasicAxisAlarms[E_BasicAxis.WriteBoolParameterError].bRaised THEN
	BasicAxisAlarms[E_BasicAxis.WriteBoolParameterError].Clear(0, 0);
END_IF

// ErrorID 15 - Command While Inhibited (WARNING)
IF ((BasicAxis.Override <= 0) AND _Busy) AND NOT BasicAxisAlarms[E_BasicAxis.CommandWhileInhibited].bRaised THEN
	RaiseAlarm(Alarm := BasicAxisAlarms[E_BasicAxis.CommandWhileInhibited]);
ELSIF NOT ((BasicAxis.Override <= 0) AND _Busy) AND BasicAxisAlarms[E_BasicAxis.CommandWhileInhibited].bRaised THEN
	BasicAxisAlarms[E_BasicAxis.CommandWhileInhibited].Clear(0, 0);
END_IF

// ErrorID 16 - NC Axis Error
IF BasicAxis.Axis.Status.Error AND NOT BasicAxisAlarms[E_BasicAxis.AxisError].bRaised THEN
	RaiseAlarmWithStrings(Alarm := BasicAxisAlarms[E_BasicAxis.AxisError], UDINT_TO_STRING(BasicAxis.Axis.Status.ErrorID), '');
ELSIF NOT BasicAxis.Axis.Status.Error AND BasicAxisAlarms[E_BasicAxis.AxisError].bRaised THEN
	BasicAxisAlarms[E_BasicAxis.AxisError].Clear(0, 0);
END_IF

// ErrorID 17 - Hardware Error
IF BasicAxis.Axis.Status.DriveDeviceError AND NOT BasicAxisAlarms[E_BasicAxis.DriveError].bRaised THEN
	RaiseAlarmWithStrings(Alarm := BasicAxisAlarms[E_BasicAxis.DriveError], UDINT_TO_STRING(18000), '');
ELSIF NOT BasicAxis.Axis.Status.DriveDeviceError AND BasicAxisAlarms[E_BasicAxis.DriveError].bRaised THEN
	BasicAxisAlarms[E_BasicAxis.DriveError].Clear(0, 0);
END_IF

// ErrorID 18 - External Sequence
IF BasicAxis.ExternalSequence <> 0 THEN
	IF (BasicAxis.ExternalSequence.Error AND NOT ExternalSequencePreviouslyErrored) AND NOT BasicAxisAlarms[E_BasicAxis.ExternalSequenceError].bRaised THEN
		ExternalSequencePreviouslyErrored := TRUE;
		RaiseAlarmWithStrings(Alarm := BasicAxisAlarms[E_BasicAxis.ExternalSequenceError], UDINT_TO_STRING(BasicAxis.ExternalSequence.ErrorID), '');
	ELSIF NOT BasicAxis.ExternalSequence.Error AND BasicAxisAlarms[E_BasicAxis.ExternalSequenceError].bRaised THEN
		BasicAxisAlarms[E_BasicAxis.ExternalSequenceError].Clear(0, 0);
	END_IF
END_IF

_CurrentAlarmSeverity := F_GetMaxSeverityRaised(Alarms := BasicAxisAlarms, CurrentSeverity := CurrentAlarmSeverity);
END_METHOD

METHOD CyclicLogic
SUPER^.CyclicLogic();
BasicAxis.CyclicLogic();
_Busy	 := BasicAxis.Busy;
_Error	 := BasicAxis.Error;
_ErrorID := BasicAxis.ErrorID;
END_METHOD

// Basic component initialization logic
METHOD PROTECTED Initialize : BOOL;

// This method is called by CyclicLogic() as required
Initialize := FALSE;
IF NOT BasicAxis.InitComplete THEN
	RETURN;
END_IF

Initialize := SUPER^.Initialize();
END_METHOD

END_FUNCTION_BLOCK

// Axes/FB_Component_BasicSlaveAxis
FUNCTION_BLOCK FB_Component_BasicSlaveAxis EXTENDS FB_ComponentBase IMPLEMENTS I_BasicSlaveAxis
VAR
	BasicSlaveAxis					  : FB_BasicSlaveAxis;
	AxisBase_HMI					  : ST_AxisBase_HMI;
	BasicAxisAlarms					  : ARRAY[1..CONSTANTS.BASIC_AXIS_ALARM_COUNT] OF FB_TcAlarm;
	BasicSlaveAxisAlarms			  : ARRAY[1..CONSTANTS.BASIC_SLAVE_AXIS_ALARM_COUNT] OF FB_TcAlarm;
	HMICommand_BasicSlaveAxis_RT	  : R_TRIG;
	ResetPreviouslyErrored			  : BOOL;
	HomePreviouslyErrored			  : BOOL;
	ExternalSequencePreviouslyErrored : BOOL;
END_VAR

// There should be no code in the function block body of a class that Implements I_CyclicFB

METHOD Disable : BOOL
Disable := BasicSlaveAxis.Disable();
END_METHOD

METHOD Enable : BOOL
Enable := BasicSlaveAxis.Enable();
END_METHOD

METHOD Home : BOOL
IF BasicSlaveAxis.Home() THEN
	HomePreviouslyErrored := FALSE;
	Home				  := TRUE;
END_IF
END_METHOD

METHOD Jog : BOOL
VAR_INPUT
	JogFW	 : BOOL;
	JogBW	 : BOOL;
	JogMode	 : E_JogMode;
	Position : LREAL;
END_VAR
Jog := BasicSlaveAxis.Jog(JogFW,
						  JogBW,
						  JogMode,
						  Position);
END_METHOD

METHOD MoveAbsolute : BOOL
VAR_INPUT
	Position	  : LREAL;
	AbortPrevious : BOOL;
END_VAR
MoveAbsolute := BasicSlaveAxis.MoveAbsolute(Position, AbortPrevious);
END_METHOD

METHOD MoveModulo : BOOL
VAR_INPUT
	Position	  : LREAL;
	Direction	  : MC_Direction;
	AbortPrevious : BOOL;
END_VAR
MoveModulo := BasicSlaveAxis.MoveModulo(Position, Direction, AbortPrevious);
END_METHOD

METHOD MoveRelative : BOOL
VAR_INPUT
	Distance	  : LREAL;
	AbortPrevious : BOOL;
END_VAR
MoveRelative := BasicSlaveAxis.MoveRelative(Distance, AbortPrevious);
END_METHOD

METHOD MoveVelocity : BOOL
VAR_INPUT
	Velocity	  : LREAL;
	AbortPrevious : BOOL;
END_VAR
MoveVelocity := BasicSlaveAxis.MoveVelocity(Velocity, AbortPrevious);
END_METHOD

METHOD ReadParameterSet : BOOL
VAR_INPUT
END_VAR
ReadParameterSet := BasicSlaveAxis.ReadParameterSet();
END_METHOD

METHOD Reset : BOOL
Reset := FALSE;
SUPER^.Reset();
IF BasicSlaveAxis.ResetMethod <> 0 THEN
	IF (BasicSlaveAxis.ResetMethod.Error AND BasicSlaveAxis.ResetPreviouslyErrored) AND BasicAxisAlarms[E_BasicAxis.ResetError].bRaised THEN
		BasicAxisAlarms[E_BasicAxis.ResetError].Clear(0, 0);
	END_IF
END_IF

IF BasicSlaveAxis.HomeMethod <> 0 THEN
	IF (BasicSlaveAxis.HomeMethod.Error AND BasicSlaveAxis.HomePreviouslyErrored) AND BasicAxisAlarms[E_BasicAxis.HomeError].bRaised THEN
		BasicAxisAlarms[E_BasicAxis.HomeError].Clear(0, 0);
	END_IF
END_IF

IF BasicSlaveAxis.ExternalSequence <> 0 THEN
	IF (BasicSlaveAxis.ExternalSequence.Error AND BasicSlaveAxis.ExternalSequencePreviouslyErrored) AND BasicAxisAlarms[E_BasicAxis.ExternalSequenceError].bRaised THEN
		BasicAxisAlarms[E_BasicAxis.ExternalSequenceError].Clear(0, 0);
	END_IF
END_IF

IF BasicSlaveAxis.Reset() THEN
	_Error				   := FALSE;
	_ErrorID			   := 0;
	ResetPreviouslyErrored := FALSE;
	Reset				   := TRUE;
END_IF
END_METHOD

METHOD RunExternalSequence : BOOL
IF BasicSlaveAxis.RunExternalSequence() THEN
	ExternalSequencePreviouslyErrored := FALSE;
	RunExternalSequence				  := TRUE;
END_IF
END_METHOD

METHOD Stop : BOOL
Stop := BasicSlaveAxis.Stop();
END_METHOD

METHOD WriteBoolParameter : BOOL
VAR_INPUT
	ParameterNumber : MC_AxisParameter;
	Value			: BOOL;
END_VAR
WriteBoolParameter := BasicSlaveAxis.WriteBoolParameter(ParameterNumber, Value);
END_METHOD

METHOD WriteParameter : BOOL
VAR_INPUT
	ParameterNumber : MC_AxisParameter;
	Value			: LREAL;
END_VAR
WriteParameter := BasicSlaveAxis.WriteParameter(ParameterNumber, Value);
END_METHOD

PROPERTY Acceleration : LREAL
GET
Acceleration := BasicSlaveAxis.Acceleration;
END_GET
SET
BasicSlaveAxis.Acceleration := Acceleration;
END_SET
END_PROPERTY

PROPERTY Deceleration : LREAL
GET
Deceleration := BasicSlaveAxis.Deceleration;
END_GET
SET
BasicSlaveAxis.Deceleration := Deceleration;
END_SET
END_PROPERTY

PROPERTY Jerk : LREAL
GET
Jerk := BasicSlaveAxis.Jerk;
END_GET
SET
BasicSlaveAxis.Jerk := Jerk;
END_SET
END_PROPERTY

PROPERTY Velocity : LREAL
GET
Velocity := BasicSlaveAxis.Velocity;
END_GET
SET
BasicSlaveAxis.Velocity := Velocity;
END_SET
END_PROPERTY

PROPERTY ActualAcceleration : LREAL
GET
ActualAcceleration := BasicSlaveAxis.ActualAcceleration;
END_GET
END_PROPERTY

PROPERTY ActualPosition : LREAL
GET
ActualPosition := BasicSlaveAxis.ActualPosition;
END_GET
END_PROPERTY

PROPERTY ActualPositionModulo : LREAL
GET
ActualPositionModulo := BasicSlaveAxis.ActualPositionModulo;
END_GET
END_PROPERTY

PROPERTY ActualTorque : LREAL
GET
ActualTorque := BasicSlaveAxis.ActualTorque;
END_GET
END_PROPERTY

PROPERTY ActualVelocity : LREAL
GET
ActualVelocity := BasicSlaveAxis.ActualVelocity;
END_GET
END_PROPERTY

PROPERTY PositionLag : LREAL
GET
PositionLag := BasicSlaveAxis.PositionLag;
END_GET
END_PROPERTY

PROPERTY SetAcceleration : LREAL
GET
SetAcceleration := BasicSlaveAxis.SetAcceleration;
END_GET
END_PROPERTY

PROPERTY SetPosition : LREAL
GET
SetPosition := BasicSlaveAxis.SetPosition;
END_GET
END_PROPERTY

PROPERTY SetPositionModulo : LREAL
GET
SetPositionModulo := BasicSlaveAxis.SetPositionModulo;
END_GET
END_PROPERTY

PROPERTY SetVelocity : LREAL
GET
SetVelocity := BasicSlaveAxis.SetVelocity;
END_GET
END_PROPERTY

PROPERTY Enabled : BOOL
GET
Enabled := BasicSlaveAxis.Enabled;
END_GET
END_PROPERTY

PROPERTY InPosition : BOOL
GET
InPosition := BasicSlaveAxis.InPosition;
END_GET
END_PROPERTY

PROPERTY Stopped : BOOL
GET
Stopped := BasicSlaveAxis.Stopped;
END_GET
END_PROPERTY

PROPERTY Axis : REFERENCE TO AXIS_REF
GET
Axis REF= BasicSlaveAxis.Axis;
END_GET
END_PROPERTY

PROPERTY AxisParameters : REFERENCE TO ST_AxisParameterSet
GET
AxisParameters REF= BasicSlaveAxis.AxisParameters;
END_GET
END_PROPERTY

PROPERTY ExternalSequence : I_MotionSequence
GET
ExternalSequence := BasicSlaveAxis.ExternalSequence;
END_GET
SET
BasicSlaveAxis.ExternalSequence := ExternalSequence;
END_SET
END_PROPERTY

PROPERTY HomeMethod : I_MotionSequence
SET
BasicSlaveAxis.HomeMethod := HomeMethod;
END_SET
END_PROPERTY

PROPERTY InhibitFeedNegative : BOOL
GET
InhibitFeedNegative := BasicSlaveAxis.InhibitFeedNegative;
END_GET
SET
BasicSlaveAxis.InhibitFeedNegative := InhibitFeedNegative;
END_SET
END_PROPERTY

PROPERTY InhibitFeedPositive : BOOL
GET
InhibitFeedPositive := BasicSlaveAxis.InhibitFeedPositive;
END_GET
SET
BasicSlaveAxis.InhibitFeedPositive := InhibitFeedPositive;
END_SET
END_PROPERTY

PROPERTY Override : LREAL
GET
Override := BasicSlaveAxis.Override;
END_GET
SET
IF Override >= 0 AND Override <= 100 THEN
	BasicSlaveAxis.Override := Override;
END_IF
END_SET
END_PROPERTY

PROPERTY ResetMethod : I_MotionSequence
GET
ResetMethod := BasicSlaveAxis.ResetMethod;
END_GET
SET
BasicSlaveAxis.ResetMethod := ResetMethod;
END_SET
END_PROPERTY

METHOD PUBLIC GearIn : BOOL
VAR_INPUT
END_VAR
GearIn := BasicSlaveAxis.GearIn();
END_METHOD

METHOD GearOut : BOOL
GearOut := BasicSlaveAxis.GearOut();
END_METHOD

PROPERTY InGear : BOOL
GET
InGear := BasicSlaveAxis.InGear;
END_GET
END_PROPERTY

PROPERTY Master1 : REFERENCE TO AXIS_REF
GET
IF __ISVALIDREF(BasicSlaveAxis.Master1) THEN
	Master1 REF= BasicSlaveAxis.Master1;
END_IF
END_GET
SET
BasicSlaveAxis.Master1 REF= Master1;
END_SET
END_PROPERTY

PROPERTY Master2 : REFERENCE TO AXIS_REF
GET
IF __ISVALIDREF(BasicSlaveAxis.Master2) THEN
	Master2 REF= BasicSlaveAxis.Master2;
END_IF
END_GET
SET
BasicSlaveAxis.Master2 REF= Master2;
END_SET
END_PROPERTY

PROPERTY Master3 : REFERENCE TO AXIS_REF
GET
IF __ISVALIDREF(BasicSlaveAxis.Master3) THEN
	Master3 REF= BasicSlaveAxis.Master3;
END_IF
END_GET
SET
BasicSlaveAxis.Master3 REF= Master3;
END_SET
END_PROPERTY

PROPERTY Master4 : REFERENCE TO AXIS_REF
GET
IF __ISVALIDREF(BasicSlaveAxis.Master4) THEN
	Master4 REF= BasicSlaveAxis.Master4;
END_IF
END_GET
SET
BasicSlaveAxis.Master4 REF= Master4;
END_SET
END_PROPERTY

PROPERTY RatioMaster1 : LREAL
GET
RatioMaster1 := BasicSlaveAxis.RatioMaster1;
END_GET
SET
BasicSlaveAxis.RatioMaster1 := RatioMaster1;
END_SET
END_PROPERTY

PROPERTY RatioMaster2 : LREAL
GET
RatioMaster2 := BasicSlaveAxis.RatioMaster2;
END_GET
SET
BasicSlaveAxis.RatioMaster2 := RatioMaster2;
END_SET
END_PROPERTY

PROPERTY RatioMaster3 : LREAL
GET
RatioMaster3 := BasicSlaveAxis.RatioMaster3;
END_GET
SET
BasicSlaveAxis.RatioMaster3 := RatioMaster3;
END_SET
END_PROPERTY

PROPERTY RatioMaster4 : LREAL
GET
RatioMaster4 := BasicSlaveAxis.RatioMaster4;
END_GET
SET
BasicSlaveAxis.RatioMaster4 := RatioMaster4;
END_SET
END_PROPERTY

METHOD PROTECTED CreateEvents
F_CreateAllEventsInClass(Alarms		:= BasicAxisAlarms,
						 ClassSize	:= SIZEOF(TC_EVENTS.BasicAxis),
						 pInitEvent := ADR(TC_EVENTS.BasicAxis.InitReferenceEvent),
						 Prefix		:= Name);

F_CreateAllEventsInClass(Alarms		:= BasicSlaveAxisAlarms,
						 ClassSize	:= SIZEOF(TC_EVENTS.BasicSlaveAxis),
						 pInitEvent := ADR(TC_EVENTS.BasicSlaveAxis.InitReferenceEvent),
						 Prefix		:= Name);

SUPER^.CreateEvents();
END_METHOD

METHOD PROTECTED HMICommunication
// Extend this method in extended FBs to communicate specific implementation data
SUPER^.HMICommunication();

// Process HMI requests

// Replace 'FALSE' below with further momentary commands (myCommand XOR myOtherCommand XOR...)
HMICommand_BasicSlaveAxis_RT(CLK := (ComponentBase_HMI.Status.HMIControlAvailable AND NOT HMICommandActive_Base) AND (FALSE));

// Signal to FB_ComponentBase that a command is active
HMICommandActive_Descendant := ComponentBase_HMI.Status.HMIControlAvailable AND (AxisBase_HMI.Command.JogFast_Backward OR AxisBase_HMI.Command.JogFast_Forward OR AxisBase_HMI.Command.JogSlow_Forward OR AxisBase_HMI.Command.JogSlow_Backward);
IF HMICommand_BasicSlaveAxis_RT.Q THEN
	;
END_IF

// Process HMI requests
IF HMICommand_BasicSlaveAxis_RT.Q THEN // If a request has been issued by the HMI, and a previous request has not just finished being processed

	//	IF AxisBaseHMI.Command.xxx THEN

	//		Enabled := TRUE;

	//	END_IF
END_IF

IF ComponentBase_HMI.Status.HMIControlAvailable AND NOT HMICommand_BasicSlaveAxis_RT.Q THEN
	IF AxisBase_HMI.Command.JogSlow_Forward THEN
		BasicSlaveAxis.Jog(AxisBase_HMI.Command.JogSlow_Forward,
						   FALSE,
						   E_JogMode.MC_JOGMODE_STANDARD_SLOW,
						   0.0);
	ELSIF AxisBase_HMI.Command.JogSlow_Backward THEN
		BasicSlaveAxis.Jog(FALSE,
						   AxisBase_HMI.Command.JogSlow_Backward,
						   E_JogMode.MC_JOGMODE_STANDARD_SLOW,
						   0.0);
	ELSIF AxisBase_HMI.Command.JogFast_Forward THEN
		BasicSlaveAxis.Jog(AxisBase_HMI.Command.JogFast_Forward,
						   FALSE,
						   E_JogMode.MC_JOGMODE_STANDARD_FAST,
						   0.0);
	ELSIF AxisBase_HMI.Command.JogFast_Backward THEN
		BasicSlaveAxis.Jog(FALSE,
						   AxisBase_HMI.Command.JogFast_Backward,
						   E_JogMode.MC_JOGMODE_STANDARD_FAST,
						   0.0);
	ELSE
		BasicSlaveAxis.Jog(FALSE,
						   FALSE,
						   E_JogMode.MC_JOGMODE_STANDARD_SLOW,
						   0.0);
	END_IF
END_IF

// Update HMI status info
AxisBase_HMI.Status.Enabled				 := BasicSlaveAxis.Enabled;
AxisBase_HMI.Status.InPosition			 := BasicSlaveAxis.InPosition;
AxisBase_HMI.Status.Stopped				 := BasicSlaveAxis.Stopped;
AxisBase_HMI.Status.Coupled				 := BasicSlaveAxis.InGear;
AxisBase_HMI.Status.SetPosition			 := BasicSlaveAxis.SetPosition;
AxisBase_HMI.Status.SetPositionModulo	 := BasicSlaveAxis.SetPositionModulo;
AxisBase_HMI.Status.SetVelocity			 := BasicSlaveAxis.SetVelocity;
AxisBase_HMI.Status.SetAcceleration		 := BasicSlaveAxis.SetAcceleration;
AxisBase_HMI.Status.ActualPosition		 := BasicSlaveAxis.ActualPosition;
AxisBase_HMI.Status.ActualPositionModulo := BasicSlaveAxis.ActualPositionModulo;
AxisBase_HMI.Status.ActualVelocity		 := BasicSlaveAxis.ActualVelocity;
AxisBase_HMI.Status.ActualAcceleration	 := BasicSlaveAxis.ActualAcceleration;
AxisBase_HMI.Status.ActualTorque		 := BasicSlaveAxis.ActualTorque;
AxisBase_HMI.Status.PositionLag			 := BasicSlaveAxis.PositionLag;
END_METHOD

METHOD PROTECTED Monitoring
SUPER^.Monitoring();

// Basic Axis Alarms

// ErrorID 2 - MC_Power
IF BasicSlaveAxis.MCPower.Error AND NOT BasicAxisAlarms[E_BasicAxis.PowerError].bRaised THEN
	RaiseAlarmWithStrings(Alarm := BasicAxisAlarms[E_BasicAxis.PowerError], UDINT_TO_STRING(BasicSlaveAxis.ErrorID), '');
ELSIF NOT BasicSlaveAxis.MCPower.Error AND BasicAxisAlarms[E_BasicAxis.PowerError].bRaised THEN
	BasicAxisAlarms[E_BasicAxis.PowerError].Clear(0, 0);
END_IF

// ErrorID 3 - MC_Reset (or other reset method)
IF BasicSlaveAxis.ResetMethod <> 0 THEN
	IF (BasicSlaveAxis.ResetMethod.Error AND NOT ResetPreviouslyErrored) AND NOT BasicAxisAlarms[E_BasicAxis.ResetError].bRaised THEN
		ResetPreviouslyErrored := TRUE;
		RaiseAlarmWithStrings(Alarm := BasicAxisAlarms[E_BasicAxis.ResetError], UDINT_TO_STRING(BasicSlaveAxis.ResetMethod.ErrorID), '');
	ELSIF NOT BasicSlaveAxis.ResetMethod.Error AND BasicAxisAlarms[E_BasicAxis.ResetError].bRaised THEN
		BasicAxisAlarms[E_BasicAxis.ResetError].Clear(0, 0);
	END_IF
END_IF

// ErrorID 4 - MC_Halt
IF BasicSlaveAxis.MCHalt.Error AND NOT BasicAxisAlarms[E_BasicAxis.HaltError].bRaised THEN
	RaiseAlarmWithStrings(Alarm := BasicAxisAlarms[E_BasicAxis.HaltError], UDINT_TO_STRING(BasicSlaveAxis.MCHalt.ErrorID), '');
ELSIF NOT BasicSlaveAxis.MCHalt.Error AND BasicAxisAlarms[E_BasicAxis.HaltError].bRaised THEN
	BasicAxisAlarms[E_BasicAxis.HaltError].Clear(0, 0);
END_IF

// ErrorID 5 - MC_Stop **NOT IMPLEMENTED**

// ErrorID 6 - MC_Home (or other home method)
IF BasicSlaveAxis.HomeMethod <> 0 THEN
	IF (BasicSlaveAxis.HomeMethod.Error AND NOT HomePreviouslyErrored) AND NOT BasicAxisAlarms[E_BasicAxis.HomeError].bRaised THEN
		HomePreviouslyErrored := TRUE;
		RaiseAlarmWithStrings(Alarm := BasicAxisAlarms[E_BasicAxis.HomeError], UDINT_TO_STRING(BasicSlaveAxis.HomeMethod.ErrorID), '');
	ELSIF NOT BasicSlaveAxis.HomeMethod.Error AND BasicAxisAlarms[E_BasicAxis.HomeError].bRaised THEN
		BasicAxisAlarms[E_BasicAxis.HomeError].Clear(0, 0);
	END_IF
END_IF

// ErrorID 7 - MC_Jog 
IF BasicSlaveAxis.MCJog.Error AND NOT BasicAxisAlarms[E_BasicAxis.JogError].bRaised THEN
	RaiseAlarmWithStrings(Alarm := BasicAxisAlarms[E_BasicAxis.JogError], UDINT_TO_STRING(BasicSlaveAxis.MCJog.ErrorID), '');
ELSIF NOT BasicSlaveAxis.MCJog.Error AND BasicAxisAlarms[E_BasicAxis.JogError].bRaised THEN
	BasicAxisAlarms[E_BasicAxis.JogError].Clear(0, 0);
END_IF

// ErrorID 8 - MC_MoveAbsolute
IF BasicSlaveAxis.MCMoveAbsolute <> 0 THEN
	IF BasicSlaveAxis.MCMoveAbsolute^.Error AND NOT BasicAxisAlarms[E_BasicAxis.MoveAbsoluteError].bRaised THEN
		RaiseAlarmWithStrings(Alarm := BasicAxisAlarms[E_BasicAxis.MoveAbsoluteError], UDINT_TO_STRING(BasicSlaveAxis.MCMoveAbsolute^.ErrorID), '');
	ELSIF NOT BasicSlaveAxis.MCMoveAbsolute^.Error AND BasicAxisAlarms[E_BasicAxis.MoveAbsoluteError].bRaised THEN
		BasicAxisAlarms[E_BasicAxis.MoveAbsoluteError].Clear(0, 0);
	END_IF
END_IF

// ErrorID 9 - MC_MoveRelative
IF BasicSlaveAxis.MCMoveRelative <> 0 THEN
	IF BasicSlaveAxis.MCMoveRelative^.Error AND NOT BasicAxisAlarms[E_BasicAxis.MoveRelativeError].bRaised THEN
		RaiseAlarmWithStrings(Alarm := BasicAxisAlarms[E_BasicAxis.MoveRelativeError], UDINT_TO_STRING(BasicSlaveAxis.MCMoveRelative^.ErrorID), '');
	ELSIF NOT BasicSlaveAxis.MCMoveRelative^.Error AND BasicAxisAlarms[E_BasicAxis.MoveRelativeError].bRaised THEN
		BasicAxisAlarms[E_BasicAxis.MoveRelativeError].Clear(0, 0);
	END_IF
END_IF

// ErrorID 10 - MC_MoveVelocity
IF BasicSlaveAxis.MCMoveVelocity <> 0 THEN
	IF BasicSlaveAxis.MCMoveVelocity^.Error AND NOT BasicAxisAlarms[E_BasicAxis.MoveVelocityError].bRaised THEN
		RaiseAlarmWithStrings(Alarm := BasicAxisAlarms[E_BasicAxis.MoveVelocityError], UDINT_TO_STRING(BasicSlaveAxis.MCMoveVelocity^.ErrorID), '');
	ELSIF NOT BasicSlaveAxis.MCMoveVelocity^.Error AND BasicAxisAlarms[E_BasicAxis.MoveVelocityError].bRaised THEN
		BasicAxisAlarms[E_BasicAxis.MoveVelocityError].Clear(0, 0);
	END_IF
END_IF

// ErrorID 11 - MC_MoveModulo
IF BasicSlaveAxis.MCMoveModulo <> 0 THEN
	IF BasicSlaveAxis.MCMoveModulo^.Error AND NOT BasicAxisAlarms[E_BasicAxis.MoveModuloError].bRaised THEN
		RaiseAlarmWithStrings(Alarm := BasicAxisAlarms[E_BasicAxis.MoveModuloError], UDINT_TO_STRING(BasicSlaveAxis.MCMoveModulo^.ErrorID), '');
	ELSIF NOT BasicSlaveAxis.MCMoveModulo^.Error AND BasicAxisAlarms[E_BasicAxis.MoveModuloError].bRaised THEN
		BasicAxisAlarms[E_BasicAxis.MoveModuloError].Clear(0, 0);
	END_IF
END_IF

// ErrorID 12 - MC_ReadParameterSet
IF BasicSlaveAxis.MCReadParameterSet.Error AND NOT BasicAxisAlarms[E_BasicAxis.ReadParameterSetError].bRaised THEN
	RaiseAlarmWithStrings(Alarm := BasicAxisAlarms[E_BasicAxis.ReadParameterSetError], UDINT_TO_STRING(BasicSlaveAxis.MCReadParameterSet.ErrorID), '');
ELSIF NOT BasicSlaveAxis.MCReadParameterSet.Error AND BasicAxisAlarms[E_BasicAxis.ReadParameterSetError].bRaised THEN
	BasicAxisAlarms[E_BasicAxis.ReadParameterSetError].Clear(0, 0);
END_IF

// ErrorID 13 - MC_WriteParameter
IF BasicSlaveAxis.MCWriteParameter.Error AND NOT BasicAxisAlarms[E_BasicAxis.WriteParameterError].bRaised THEN
	RaiseAlarmWithStrings(Alarm := BasicAxisAlarms[E_BasicAxis.WriteParameterError], UDINT_TO_STRING(BasicSlaveAxis.MCWriteParameter.ErrorID), '');
ELSIF NOT BasicSlaveAxis.MCWriteParameter.Error AND BasicAxisAlarms[E_BasicAxis.WriteParameterError].bRaised THEN
	BasicAxisAlarms[E_BasicAxis.WriteParameterError].Clear(0, 0);
END_IF

// ErrorID 14 - MC_WriteBoolParameter
IF BasicSlaveAxis.MCWriteBoolParameter.Error AND NOT BasicAxisAlarms[E_BasicAxis.WriteBoolParameterError].bRaised THEN
	RaiseAlarmWithStrings(Alarm := BasicAxisAlarms[E_BasicAxis.WriteBoolParameterError], UDINT_TO_STRING(BasicSlaveAxis.MCWriteBoolParameter.ErrorID), '');
ELSIF NOT BasicSlaveAxis.MCWriteBoolParameter.Error AND BasicAxisAlarms[E_BasicAxis.WriteBoolParameterError].bRaised THEN
	BasicAxisAlarms[E_BasicAxis.WriteBoolParameterError].Clear(0, 0);
END_IF

// ErrorID 15 - Command While Inhibited (WARNING)
IF ((BasicSlaveAxis.Override <= 0) AND _Busy) AND NOT BasicAxisAlarms[E_BasicAxis.CommandWhileInhibited].bRaised THEN
	RaiseAlarm(Alarm := BasicAxisAlarms[E_BasicAxis.CommandWhileInhibited]);
ELSIF NOT ((BasicSlaveAxis.Override <= 0) AND _Busy) AND BasicAxisAlarms[E_BasicAxis.CommandWhileInhibited].bRaised THEN
	BasicAxisAlarms[E_BasicAxis.CommandWhileInhibited].Clear(0, 0);
END_IF

// ErrorID 16 - NC Axis Error
IF BasicSlaveAxis.Axis.Status.Error AND NOT BasicAxisAlarms[E_BasicAxis.AxisError].bRaised THEN
	RaiseAlarmWithStrings(Alarm := BasicAxisAlarms[E_BasicAxis.AxisError], UDINT_TO_STRING(BasicSlaveAxis.Axis.Status.ErrorID), '');
ELSIF NOT BasicSlaveAxis.Axis.Status.Error AND BasicAxisAlarms[E_BasicAxis.AxisError].bRaised THEN
	BasicAxisAlarms[E_BasicAxis.AxisError].Clear(0, 0);
END_IF

// ErrorID 17 - Hardware Error
IF BasicSlaveAxis.Axis.Status.DriveDeviceError AND NOT BasicAxisAlarms[E_BasicAxis.DriveError].bRaised THEN
	RaiseAlarmWithStrings(Alarm := BasicAxisAlarms[E_BasicAxis.DriveError], UDINT_TO_STRING(18000), '');
ELSIF NOT BasicSlaveAxis.Axis.Status.DriveDeviceError AND BasicAxisAlarms[E_BasicAxis.DriveError].bRaised THEN
	BasicAxisAlarms[E_BasicAxis.DriveError].Clear(0, 0);
END_IF

// ErrorID 18 - External Sequence
IF BasicSlaveAxis.ExternalSequence <> 0 THEN
	IF (BasicSlaveAxis.ExternalSequence.Error AND NOT ExternalSequencePreviouslyErrored) AND NOT BasicAxisAlarms[E_BasicAxis.ExternalSequenceError].bRaised THEN
		ExternalSequencePreviouslyErrored := TRUE;
		RaiseAlarmWithStrings(Alarm := BasicAxisAlarms[E_BasicAxis.ExternalSequenceError], UDINT_TO_STRING(BasicSlaveAxis.ExternalSequence.ErrorID), '');
	ELSIF NOT BasicSlaveAxis.ExternalSequence.Error AND BasicAxisAlarms[E_BasicAxis.ExternalSequenceError].bRaised THEN
		BasicAxisAlarms[E_BasicAxis.ExternalSequenceError].Clear(0, 0);
	END_IF
END_IF

// Basic Slave Axis Alarms

// ErrorID 2 - MC_GearInMultimaster
IF BasicSlaveAxis.MCGearInMultimaster.Error AND NOT BasicAxisAlarms[E_BasicSlaveAxis.GearInMultimasterError].bRaised THEN
	RaiseAlarmWithStrings(Alarm := BasicSlaveAxisAlarms[E_BasicSlaveAxis.GearInMultimasterError], UDINT_TO_STRING(BasicSlaveAxis.MCGearInMultimaster.ErrorID), '');
ELSIF NOT BasicSlaveAxis.MCGearInMultimaster.Error AND BasicSlaveAxisAlarms[E_BasicSlaveAxis.GearInMultimasterError].bRaised THEN
	BasicSlaveAxisAlarms[E_BasicSlaveAxis.GearInMultimasterError].Clear(0, 0);
END_IF

// ErrorID 3 - MC_GearOut
IF BasicSlaveAxis.MCGearOut.Error AND NOT BasicAxisAlarms[E_BasicSlaveAxis.GearOutError].bRaised THEN
	RaiseAlarmWithStrings(Alarm := BasicSlaveAxisAlarms[E_BasicSlaveAxis.GearOutError], UDINT_TO_STRING(BasicSlaveAxis.MCGearOut.ErrorID), '');
ELSIF NOT BasicSlaveAxis.MCGearOut.Error AND BasicSlaveAxisAlarms[E_BasicSlaveAxis.GearOutError].bRaised THEN
	BasicSlaveAxisAlarms[E_BasicSlaveAxis.GearOutError].Clear(0, 0);
END_IF

_CurrentAlarmSeverity := F_GetMaxSeverityRaised(Alarms := BasicAxisAlarms, CurrentSeverity := CurrentAlarmSeverity);
_CurrentAlarmSeverity := F_GetMaxSeverityRaised(Alarms := BasicSlaveAxisAlarms, CurrentSeverity := CurrentAlarmSeverity);
END_METHOD

METHOD CyclicLogic
SUPER^.CyclicLogic();
BasicSlaveAxis.CyclicLogic();
_Busy	 := BasicSlaveAxis.Busy;
_Error	 := BasicSlaveAxis.Error;
_ErrorID := BasicSlaveAxis.ErrorID;
END_METHOD

// Basic component initialization logic
METHOD PROTECTED Initialize : BOOL;

// This method is called by CyclicLogic() as required
IF NOT BasicSlaveAxis.InitComplete THEN
	RETURN;
END_IF

Initialize := SUPER^.Initialize();
END_METHOD

END_FUNCTION_BLOCK

// Axes/FB_Component_CamSlaveAxis
FUNCTION_BLOCK FB_Component_CamSlaveAxis EXTENDS FB_ComponentBase IMPLEMENTS I_CamSlaveAxis
VAR
	CamSlaveAxis					  : FB_CamSlaveAxis;
	AxisBase_HMI					  : ST_AxisBase_HMI;
	BasicAxisAlarms					  : ARRAY[1..CONSTANTS.BASIC_AXIS_ALARM_COUNT] OF FB_TcAlarm;
	CamSlaveAxisAlarms				  : ARRAY[1..CONSTANTS.CAM_SLAVE_AXIS_ALARM_COUNT] OF FB_TcAlarm;
	HMICommand_CamSlaveAxis_RT		  : R_TRIG;
	ResetPreviouslyErrored			  : BOOL;
	HomePreviouslyErrored			  : BOOL;
	ExternalSequencePreviouslyErrored : BOOL;
END_VAR

// There should be no code in the function block body of a class that Implements I_CyclicFB

METHOD Disable : BOOL
Disable := CamSlaveAxis.Disable();
END_METHOD

METHOD Enable : BOOL
Enable := CamSlaveAxis.Enable();
END_METHOD

METHOD Home : BOOL
IF CamSlaveAxis.Home() THEN
	HomePreviouslyErrored := FALSE;
	Home				  := TRUE;
END_IF
END_METHOD

METHOD Jog : BOOL
VAR_INPUT
	JogFW	 : BOOL;
	JogBW	 : BOOL;
	JogMode	 : E_JogMode;
	Position : LREAL;
END_VAR
Jog := CamSlaveAxis.Jog(JogFW,
						JogBW,
						JogMode,
						Position);
END_METHOD

METHOD MoveAbsolute : BOOL
VAR_INPUT
	Position	  : LREAL;
	AbortPrevious : BOOL;
END_VAR
MoveAbsolute := CamSlaveAxis.MoveAbsolute(Position, AbortPrevious);
END_METHOD

METHOD MoveModulo : BOOL
VAR_INPUT
	Position	  : LREAL;
	Direction	  : MC_Direction;
	AbortPrevious : BOOL;
END_VAR
MoveModulo := CamSlaveAxis.MoveModulo(Position, Direction, AbortPrevious);
END_METHOD

METHOD MoveRelative : BOOL
VAR_INPUT
	Distance	  : LREAL;
	AbortPrevious : BOOL;
END_VAR
MoveRelative := CamSlaveAxis.MoveRelative(Distance, AbortPrevious);
END_METHOD

METHOD MoveVelocity : BOOL
VAR_INPUT
	Velocity	  : LREAL;
	AbortPrevious : BOOL;
END_VAR
MoveVelocity := CamSlaveAxis.MoveVelocity(Velocity, AbortPrevious);
END_METHOD

METHOD ReadParameterSet : BOOL
VAR_INPUT
END_VAR
ReadParameterSet := CamSlaveAxis.ReadParameterSet();
END_METHOD

METHOD Reset : BOOL
Reset := FALSE;
SUPER^.Reset();
IF CamSlaveAxis.ResetMethod <> 0 THEN
	IF (CamSlaveAxis.ResetMethod.Error AND CamSlaveAxis.ResetPreviouslyErrored) AND BasicAxisAlarms[E_BasicAxis.ResetError].bRaised THEN
		BasicAxisAlarms[E_BasicAxis.ResetError].Clear(0, 0);
	END_IF
END_IF

IF CamSlaveAxis.HomeMethod <> 0 THEN
	IF (CamSlaveAxis.HomeMethod.Error AND CamSlaveAxis.HomePreviouslyErrored) AND BasicAxisAlarms[E_BasicAxis.HomeError].bRaised THEN
		BasicAxisAlarms[E_BasicAxis.HomeError].Clear(0, 0);
	END_IF
END_IF

IF CamSlaveAxis.ExternalSequence <> 0 THEN
	IF (CamSlaveAxis.ExternalSequence.Error AND CamSlaveAxis.ExternalSequencePreviouslyErrored) AND BasicAxisAlarms[E_BasicAxis.ExternalSequenceError].bRaised THEN
		BasicAxisAlarms[E_BasicAxis.ExternalSequenceError].Clear(0, 0);
	END_IF
END_IF

IF CamSlaveAxis.Reset() THEN
	_Error				   := FALSE;
	_ErrorID			   := 0;
	ResetPreviouslyErrored := FALSE;
	Reset				   := TRUE;
END_IF
END_METHOD

METHOD RunExternalSequence : BOOL
IF CamSlaveAxis.RunExternalSequence() THEN
	ExternalSequencePreviouslyErrored := FALSE;
	RunExternalSequence				  := TRUE;
END_IF
END_METHOD

METHOD Stop : BOOL
Stop := CamSlaveAxis.Stop();
END_METHOD

METHOD WriteBoolParameter : BOOL
VAR_INPUT
	ParameterNumber : MC_AxisParameter;
	Value			: BOOL;
END_VAR
WriteBoolParameter := CamSlaveAxis.WriteBoolParameter(ParameterNumber, Value);
END_METHOD

METHOD WriteParameter : BOOL
VAR_INPUT
	ParameterNumber : MC_AxisParameter;
	Value			: LREAL;
END_VAR
WriteParameter := CamSlaveAxis.WriteParameter(ParameterNumber, Value);
END_METHOD

PROPERTY Acceleration : LREAL
GET
Acceleration := CamSlaveAxis.Acceleration;
END_GET
SET
CamSlaveAxis.Acceleration := Acceleration;
END_SET
END_PROPERTY

PROPERTY Deceleration : LREAL
GET
Deceleration := CamSlaveAxis.Deceleration;
END_GET
SET
CamSlaveAxis.Deceleration := Deceleration;
END_SET
END_PROPERTY

PROPERTY Jerk : LREAL
GET
Jerk := CamSlaveAxis.Jerk;
END_GET
SET
CamSlaveAxis.Jerk := Jerk;
END_SET
END_PROPERTY

PROPERTY Velocity : LREAL
GET
Velocity := CamSlaveAxis.Velocity;
END_GET
SET
CamSlaveAxis.Velocity := Velocity;
END_SET
END_PROPERTY

PROPERTY ActualAcceleration : LREAL
GET
ActualAcceleration := CamSlaveAxis.ActualAcceleration;
END_GET
END_PROPERTY

PROPERTY ActualPosition : LREAL
GET
ActualPosition := CamSlaveAxis.ActualPosition;
END_GET
END_PROPERTY

PROPERTY ActualPositionModulo : LREAL
GET
ActualPositionModulo := CamSlaveAxis.ActualPositionModulo;
END_GET
END_PROPERTY

PROPERTY ActualTorque : LREAL
GET
ActualTorque := CamSlaveAxis.ActualTorque;
END_GET
END_PROPERTY

PROPERTY ActualVelocity : LREAL
GET
ActualVelocity := CamSlaveAxis.ActualVelocity;
END_GET
END_PROPERTY

PROPERTY PositionLag : LREAL
GET
PositionLag := CamSlaveAxis.PositionLag;
END_GET
END_PROPERTY

PROPERTY SetAcceleration : LREAL
GET
SetAcceleration := CamSlaveAxis.SetAcceleration;
END_GET
END_PROPERTY

PROPERTY SetPosition : LREAL
GET
SetPosition := CamSlaveAxis.SetPosition;
END_GET
END_PROPERTY

PROPERTY SetPositionModulo : LREAL
GET
SetPositionModulo := CamSlaveAxis.SetPositionModulo;
END_GET
END_PROPERTY

PROPERTY SetVelocity : LREAL
GET
SetVelocity := CamSlaveAxis.SetVelocity;
END_GET
END_PROPERTY

PROPERTY Enabled : BOOL
GET
Enabled := CamSlaveAxis.Enabled;
END_GET
END_PROPERTY

PROPERTY InPosition : BOOL
GET
InPosition := CamSlaveAxis.InPosition;
END_GET
END_PROPERTY

PROPERTY Stopped : BOOL
GET
Stopped := CamSlaveAxis.Stopped;
END_GET
END_PROPERTY

PROPERTY Axis : REFERENCE TO AXIS_REF
GET
Axis REF= CamSlaveAxis.Axis;
END_GET
END_PROPERTY

PROPERTY AxisParameters : REFERENCE TO ST_AxisParameterSet
GET
AxisParameters REF= CamSlaveAxis.AxisParameters;
END_GET
END_PROPERTY

PROPERTY ExternalSequence : I_MotionSequence
GET
ExternalSequence := CamSlaveAxis.ExternalSequence;
END_GET
SET
CamSlaveAxis.ExternalSequence := ExternalSequence;
END_SET
END_PROPERTY

PROPERTY HomeMethod : I_MotionSequence
SET
CamSlaveAxis.HomeMethod := HomeMethod;
END_SET
END_PROPERTY

PROPERTY InhibitFeedNegative : BOOL
GET
InhibitFeedNegative := CamSlaveAxis.InhibitFeedNegative;
END_GET
SET
CamSlaveAxis.InhibitFeedNegative := InhibitFeedNegative;
END_SET
END_PROPERTY

PROPERTY InhibitFeedPositive : BOOL
GET
InhibitFeedPositive := CamSlaveAxis.InhibitFeedPositive;
END_GET
SET
CamSlaveAxis.InhibitFeedPositive := InhibitFeedPositive;
END_SET
END_PROPERTY

PROPERTY Override : LREAL
GET
Override := CamSlaveAxis.Override;
END_GET
SET
IF Override >= 0 AND Override <= 100 THEN
	CamSlaveAxis.Override := Override;
END_IF
END_SET
END_PROPERTY

PROPERTY ResetMethod : I_MotionSequence
GET
ResetMethod := CamSlaveAxis.ResetMethod;
END_GET
SET
CamSlaveAxis.ResetMethod := ResetMethod;
END_SET
END_PROPERTY

PROPERTY CamParameters : REFERENCE TO ST_CamParameters
GET
IF __ISVALIDREF(CamSlaveAxis._CamParameters) THEN
	CamParameters REF= CamSlaveAxis._CamParameters;
END_IF
END_GET
SET
CamSlaveAxis.CamParameters REF= CamParameters;
END_SET
END_PROPERTY

METHOD ChangeMode : BOOL
VAR_INPUT
END_VAR
ChangeMode := CamSlaveAxis.ChangeMode();
END_METHOD

METHOD FindSlavePos : BOOL
VAR_INPUT
END_VAR
FindSlavePos := CamSlaveAxis.FindSlavePos();
END_METHOD

METHOD FindSyncPos : BOOL
VAR_INPUT
END_VAR
FindSyncPos := CamSlaveAxis.FindSyncPos();
END_METHOD

PROPERTY InSync : BOOL
GET
InSync := CamSlaveAxis._InSync;
END_GET
END_PROPERTY

PROPERTY Master : REFERENCE TO Tc2_MC2.AXIS_REF
GET
IF __ISVALIDREF(CamSlaveAxis.Master) THEN
	Master REF= CamSlaveAxis.Master;
END_IF
END_GET
SET
CamSlaveAxis.Master REF= Master;
END_SET
END_PROPERTY

PROPERTY RunningTable : UDINT
GET
RunningTable := CamSlaveAxis._RunningTable;
END_GET
END_PROPERTY

METHOD StartCouple : BOOL
VAR_INPUT
END_VAR
StartCouple := CamSlaveAxis.StartCouple();
END_METHOD

METHOD StartSync : BOOL
VAR_INPUT
END_VAR
StartSync := CamSlaveAxis.StartSync();
END_METHOD

PROPERTY SyncPos : LREAL
GET
SyncPos := CamSlaveAxis._SyncPos;
END_GET
END_PROPERTY

METHOD UpdateTable : BOOL
VAR_INPUT
END_VAR
UpdateTable := CamSlaveAxis.UpdateTable();
END_METHOD

//Check before calling: FindSlavePosition, FindSyncPosition, StartSync
PROPERTY WaitingForCommand : BOOL
GET
WaitingForCommand := CamSlaveAxis.WaitingForCommand;
END_GET
END_PROPERTY

METHOD PROTECTED CreateEvents
F_CreateAllEventsInClass(Alarms		:= BasicAxisAlarms,
						 ClassSize	:= SIZEOF(TC_EVENTS.BasicAxis),
						 pInitEvent := ADR(TC_EVENTS.BasicAxis.InitReferenceEvent),
						 Prefix		:= Name);

F_CreateAllEventsInClass(Alarms		:= CamSlaveAxisAlarms,
						 ClassSize	:= SIZEOF(TC_EVENTS.CamSlaveAxis),
						 pInitEvent := ADR(TC_EVENTS.CamSlaveAxis.InitReferenceEvent),
						 Prefix		:= Name);

SUPER^.CreateEvents();
END_METHOD

METHOD PROTECTED HMICommunication
// Extend this method in extended FBs to communicate specific implementation data
SUPER^.HMICommunication();

// Process HMI requests

// Replace 'FALSE' below with further momentary commands (myCommand XOR myOtherCommand XOR...)
HMICommand_CamSlaveAxis_RT(CLK := (ComponentBase_HMI.Status.HMIControlAvailable AND NOT HMICommandActive_Base) AND (FALSE));

// Signal to FB_ComponentBase that a command is active
HMICommandActive_Descendant := ComponentBase_HMI.Status.HMIControlAvailable AND (AxisBase_HMI.Command.JogFast_Backward OR AxisBase_HMI.Command.JogFast_Forward OR AxisBase_HMI.Command.JogSlow_Forward OR AxisBase_HMI.Command.JogSlow_Backward);
IF HMICommand_CamSlaveAxis_RT.Q THEN
	;
END_IF

// Process HMI requests
IF HMICommand_CamSlaveAxis_RT.Q THEN // If a request has been issued by the HMI, and a previous request has not just finished being processed

	//	IF AxisBaseHMI.Command.xxx THEN

	//		Enabled := TRUE;

	//	END_IF
END_IF

IF ComponentBase_HMI.Status.HMIControlAvailable AND NOT HMICommand_CamSlaveAxis_RT.Q THEN
	IF AxisBase_HMI.Command.JogSlow_Forward THEN
		CamSlaveAxis.Jog(AxisBase_HMI.Command.JogSlow_Forward,
						 FALSE,
						 E_JogMode.MC_JOGMODE_STANDARD_SLOW,
						 0.0);
	ELSIF AxisBase_HMI.Command.JogSlow_Backward THEN
		CamSlaveAxis.Jog(FALSE,
						 AxisBase_HMI.Command.JogSlow_Backward,
						 E_JogMode.MC_JOGMODE_STANDARD_SLOW,
						 0.0);
	ELSIF AxisBase_HMI.Command.JogFast_Forward THEN
		CamSlaveAxis.Jog(AxisBase_HMI.Command.JogFast_Forward,
						 FALSE,
						 E_JogMode.MC_JOGMODE_STANDARD_FAST,
						 0.0);
	ELSIF AxisBase_HMI.Command.JogFast_Backward THEN
		CamSlaveAxis.Jog(FALSE,
						 AxisBase_HMI.Command.JogFast_Backward,
						 E_JogMode.MC_JOGMODE_STANDARD_FAST,
						 0.0);
	ELSE
		CamSlaveAxis.Jog(FALSE,
						 FALSE,
						 E_JogMode.MC_JOGMODE_STANDARD_SLOW,
						 0.0);
	END_IF
END_IF

// Update HMI status info
AxisBase_HMI.Status.Enabled				 := CamSlaveAxis.Enabled;
AxisBase_HMI.Status.InPosition			 := CamSlaveAxis.InPosition;
AxisBase_HMI.Status.Stopped				 := CamSlaveAxis.Stopped;
AxisBase_HMI.Status.Coupled				 := CamSlaveAxis.InSync;
AxisBase_HMI.Status.SetPosition			 := CamSlaveAxis.SetPosition;
AxisBase_HMI.Status.SetPositionModulo	 := CamSlaveAxis.SetPositionModulo;
AxisBase_HMI.Status.SetVelocity			 := CamSlaveAxis.SetVelocity;
AxisBase_HMI.Status.SetAcceleration		 := CamSlaveAxis.SetAcceleration;
AxisBase_HMI.Status.ActualPosition		 := CamSlaveAxis.ActualPosition;
AxisBase_HMI.Status.ActualPositionModulo := CamSlaveAxis.ActualPositionModulo;
AxisBase_HMI.Status.ActualVelocity		 := CamSlaveAxis.ActualVelocity;
AxisBase_HMI.Status.ActualAcceleration	 := CamSlaveAxis.ActualAcceleration;
AxisBase_HMI.Status.ActualTorque		 := CamSlaveAxis.ActualTorque;
AxisBase_HMI.Status.PositionLag			 := CamSlaveAxis.PositionLag;
END_METHOD

METHOD PROTECTED Monitoring
SUPER^.Monitoring();

// Basic Axis Alarms

// ErrorID 2 - MC_Power
IF CamSlaveAxis.MCPower.Error AND NOT BasicAxisAlarms[E_BasicAxis.PowerError].bRaised THEN
	RaiseAlarmWithStrings(Alarm := BasicAxisAlarms[E_BasicAxis.PowerError], UDINT_TO_STRING(CamSlaveAxis.ErrorID), '');
ELSIF NOT CamSlaveAxis.MCPower.Error AND BasicAxisAlarms[E_BasicAxis.PowerError].bRaised THEN
	BasicAxisAlarms[E_BasicAxis.PowerError].Clear(0, 0);
END_IF

// ErrorID 3 - MC_Reset (or other reset method)
IF CamSlaveAxis.ResetMethod <> 0 THEN
	IF (CamSlaveAxis.ResetMethod.Error AND NOT ResetPreviouslyErrored) AND NOT BasicAxisAlarms[E_BasicAxis.ResetError].bRaised THEN
		ResetPreviouslyErrored := TRUE;
		RaiseAlarmWithStrings(Alarm := BasicAxisAlarms[E_BasicAxis.ResetError], UDINT_TO_STRING(CamSlaveAxis.ResetMethod.ErrorID), '');
	ELSIF NOT CamSlaveAxis.ResetMethod.Error AND BasicAxisAlarms[E_BasicAxis.ResetError].bRaised THEN
		BasicAxisAlarms[E_BasicAxis.ResetError].Clear(0, 0);
	END_IF
END_IF

// ErrorID 4 - MC_Halt
IF CamSlaveAxis.MCHalt.Error AND NOT BasicAxisAlarms[E_BasicAxis.HaltError].bRaised THEN
	RaiseAlarmWithStrings(Alarm := BasicAxisAlarms[E_BasicAxis.HaltError], UDINT_TO_STRING(CamSlaveAxis.MCHalt.ErrorID), '');
ELSIF NOT CamSlaveAxis.MCHalt.Error AND BasicAxisAlarms[E_BasicAxis.HaltError].bRaised THEN
	BasicAxisAlarms[E_BasicAxis.HaltError].Clear(0, 0);
END_IF

// ErrorID 5 - MC_Stop **NOT IMPLEMENTED**

// ErrorID 6 - MC_Home (or other home method)
IF CamSlaveAxis.HomeMethod <> 0 THEN
	IF (CamSlaveAxis.HomeMethod.Error AND NOT HomePreviouslyErrored) AND NOT BasicAxisAlarms[E_BasicAxis.HomeError].bRaised THEN
		HomePreviouslyErrored := TRUE;
		RaiseAlarmWithStrings(Alarm := BasicAxisAlarms[E_BasicAxis.HomeError], UDINT_TO_STRING(CamSlaveAxis.HomeMethod.ErrorID), '');
	ELSIF NOT CamSlaveAxis.HomeMethod.Error AND BasicAxisAlarms[E_BasicAxis.HomeError].bRaised THEN
		BasicAxisAlarms[E_BasicAxis.HomeError].Clear(0, 0);
	END_IF
END_IF

// ErrorID 7 - MC_Jog 
IF CamSlaveAxis.MCJog.Error AND NOT BasicAxisAlarms[E_BasicAxis.JogError].bRaised THEN
	RaiseAlarmWithStrings(Alarm := BasicAxisAlarms[E_BasicAxis.JogError], UDINT_TO_STRING(CamSlaveAxis.MCJog.ErrorID), '');
ELSIF NOT CamSlaveAxis.MCJog.Error AND BasicAxisAlarms[E_BasicAxis.JogError].bRaised THEN
	BasicAxisAlarms[E_BasicAxis.JogError].Clear(0, 0);
END_IF

// ErrorID 8 - MC_MoveAbsolute
IF CamSlaveAxis.MCMoveAbsolute <> 0 THEN
	IF CamSlaveAxis.MCMoveAbsolute^.Error AND NOT BasicAxisAlarms[E_BasicAxis.MoveAbsoluteError].bRaised THEN
		RaiseAlarmWithStrings(Alarm := BasicAxisAlarms[E_BasicAxis.MoveAbsoluteError], UDINT_TO_STRING(CamSlaveAxis.MCMoveAbsolute^.ErrorID), '');
	ELSIF NOT CamSlaveAxis.MCMoveAbsolute^.Error AND BasicAxisAlarms[E_BasicAxis.MoveAbsoluteError].bRaised THEN
		BasicAxisAlarms[E_BasicAxis.MoveAbsoluteError].Clear(0, 0);
	END_IF
END_IF

// ErrorID 9 - MC_MoveRelative
IF CamSlaveAxis.MCMoveRelative <> 0 THEN
	IF CamSlaveAxis.MCMoveRelative^.Error AND NOT BasicAxisAlarms[E_BasicAxis.MoveRelativeError].bRaised THEN
		RaiseAlarmWithStrings(Alarm := BasicAxisAlarms[E_BasicAxis.MoveRelativeError], UDINT_TO_STRING(CamSlaveAxis.MCMoveRelative^.ErrorID), '');
	ELSIF NOT CamSlaveAxis.MCMoveRelative^.Error AND BasicAxisAlarms[E_BasicAxis.MoveRelativeError].bRaised THEN
		BasicAxisAlarms[E_BasicAxis.MoveRelativeError].Clear(0, 0);
	END_IF
END_IF

// ErrorID 10 - MC_MoveVelocity
IF CamSlaveAxis.MCMoveVelocity <> 0 THEN
	IF CamSlaveAxis.MCMoveVelocity^.Error AND NOT BasicAxisAlarms[E_BasicAxis.MoveVelocityError].bRaised THEN
		RaiseAlarmWithStrings(Alarm := BasicAxisAlarms[E_BasicAxis.MoveVelocityError], UDINT_TO_STRING(CamSlaveAxis.MCMoveVelocity^.ErrorID), '');
	ELSIF NOT CamSlaveAxis.MCMoveVelocity^.Error AND BasicAxisAlarms[E_BasicAxis.MoveVelocityError].bRaised THEN
		BasicAxisAlarms[E_BasicAxis.MoveVelocityError].Clear(0, 0);
	END_IF
END_IF

// ErrorID 11 - MC_MoveModulo
IF CamSlaveAxis.MCMoveModulo <> 0 THEN
	IF CamSlaveAxis.MCMoveModulo^.Error AND NOT BasicAxisAlarms[E_BasicAxis.MoveModuloError].bRaised THEN
		RaiseAlarmWithStrings(Alarm := BasicAxisAlarms[E_BasicAxis.MoveModuloError], UDINT_TO_STRING(CamSlaveAxis.MCMoveModulo^.ErrorID), '');
	ELSIF NOT CamSlaveAxis.MCMoveModulo^.Error AND BasicAxisAlarms[E_BasicAxis.MoveModuloError].bRaised THEN
		BasicAxisAlarms[E_BasicAxis.MoveModuloError].Clear(0, 0);
	END_IF
END_IF

// ErrorID 12 - MC_ReadParameterSet
IF CamSlaveAxis.MCReadParameterSet.Error AND NOT BasicAxisAlarms[E_BasicAxis.ReadParameterSetError].bRaised THEN
	RaiseAlarmWithStrings(Alarm := BasicAxisAlarms[E_BasicAxis.ReadParameterSetError], UDINT_TO_STRING(CamSlaveAxis.MCReadParameterSet.ErrorID), '');
ELSIF NOT CamSlaveAxis.MCReadParameterSet.Error AND BasicAxisAlarms[E_BasicAxis.ReadParameterSetError].bRaised THEN
	BasicAxisAlarms[E_BasicAxis.ReadParameterSetError].Clear(0, 0);
END_IF

// ErrorID 13 - MC_WriteParameter
IF CamSlaveAxis.MCWriteParameter.Error AND NOT BasicAxisAlarms[E_BasicAxis.WriteParameterError].bRaised THEN
	RaiseAlarmWithStrings(Alarm := BasicAxisAlarms[E_BasicAxis.WriteParameterError], UDINT_TO_STRING(CamSlaveAxis.MCWriteParameter.ErrorID), '');
ELSIF NOT CamSlaveAxis.MCWriteParameter.Error AND BasicAxisAlarms[E_BasicAxis.WriteParameterError].bRaised THEN
	BasicAxisAlarms[E_BasicAxis.WriteParameterError].Clear(0, 0);
END_IF

// ErrorID 14 - MC_WriteBoolParameter
IF CamSlaveAxis.MCWriteBoolParameter.Error AND NOT BasicAxisAlarms[E_BasicAxis.WriteBoolParameterError].bRaised THEN
	RaiseAlarmWithStrings(Alarm := BasicAxisAlarms[E_BasicAxis.WriteBoolParameterError], UDINT_TO_STRING(CamSlaveAxis.MCWriteBoolParameter.ErrorID), '');
ELSIF NOT CamSlaveAxis.MCWriteBoolParameter.Error AND BasicAxisAlarms[E_BasicAxis.WriteBoolParameterError].bRaised THEN
	BasicAxisAlarms[E_BasicAxis.WriteBoolParameterError].Clear(0, 0);
END_IF

// ErrorID 15 - Command While Inhibited (WARNING)
IF ((CamSlaveAxis.Override <= 0) AND _Busy) AND NOT BasicAxisAlarms[E_BasicAxis.CommandWhileInhibited].bRaised THEN
	RaiseAlarm(Alarm := BasicAxisAlarms[E_BasicAxis.CommandWhileInhibited]);
ELSIF NOT ((CamSlaveAxis.Override <= 0) AND _Busy) AND BasicAxisAlarms[E_BasicAxis.CommandWhileInhibited].bRaised THEN
	BasicAxisAlarms[E_BasicAxis.CommandWhileInhibited].Clear(0, 0);
END_IF

// ErrorID 16 - NC Axis Error
IF CamSlaveAxis.Axis.Status.Error AND NOT BasicAxisAlarms[E_BasicAxis.AxisError].bRaised THEN
	RaiseAlarmWithStrings(Alarm := BasicAxisAlarms[E_BasicAxis.AxisError], UDINT_TO_STRING(CamSlaveAxis.Axis.Status.ErrorID), '');
ELSIF NOT CamSlaveAxis.Axis.Status.Error AND BasicAxisAlarms[E_BasicAxis.AxisError].bRaised THEN
	BasicAxisAlarms[E_BasicAxis.AxisError].Clear(0, 0);
END_IF

// ErrorID 17 - Hardware Error
IF CamSlaveAxis.Axis.Status.DriveDeviceError AND NOT BasicAxisAlarms[E_BasicAxis.DriveError].bRaised THEN
	RaiseAlarmWithStrings(Alarm := BasicAxisAlarms[E_BasicAxis.DriveError], UDINT_TO_STRING(18000), '');
ELSIF NOT CamSlaveAxis.Axis.Status.DriveDeviceError AND BasicAxisAlarms[E_BasicAxis.DriveError].bRaised THEN
	BasicAxisAlarms[E_BasicAxis.DriveError].Clear(0, 0);
END_IF

// ErrorID 18 - External Sequence
IF CamSlaveAxis.ExternalSequence <> 0 THEN
	IF (CamSlaveAxis.ExternalSequence.Error AND NOT ExternalSequencePreviouslyErrored) AND NOT BasicAxisAlarms[E_BasicAxis.ExternalSequenceError].bRaised THEN
		ExternalSequencePreviouslyErrored := TRUE;
		RaiseAlarmWithStrings(Alarm := BasicAxisAlarms[E_BasicAxis.ExternalSequenceError], UDINT_TO_STRING(CamSlaveAxis.ExternalSequence.ErrorID), '');
	ELSIF NOT CamSlaveAxis.ExternalSequence.Error AND BasicAxisAlarms[E_BasicAxis.ExternalSequenceError].bRaised THEN
		BasicAxisAlarms[E_BasicAxis.ExternalSequenceError].Clear(0, 0);
	END_IF
END_IF

// ErrorID 2 - MC_CamIn
IF CamSlaveAxis.McCamIn.Error AND NOT CamSlaveAxisAlarms[E_CamSlaveAxis.McCamInError].bRaised THEN
	RaiseAlarmWithStrings(Alarm := CamSlaveAxisAlarms[E_CamSlaveAxis.McCamInError], UDINT_TO_STRING(CamSlaveAxis.ErrorID), '');
ELSIF NOT CamSlaveAxis.McCamIn.Error AND CamSlaveAxisAlarms[E_CamSlaveAxis.McCamInError].bRaised THEN
	CamSlaveAxisAlarms[E_CamSlaveAxis.McCamInError].Clear(0, 0);
END_IF

// ErrorID 3 - MC_CamOut
IF CamSlaveAxis.McCamOut.Error AND NOT CamSlaveAxisAlarms[E_CamSlaveAxis.McCamOutError].bRaised THEN
	RaiseAlarmWithStrings(Alarm := CamSlaveAxisAlarms[E_CamSlaveAxis.McCamOutError], UDINT_TO_STRING(CamSlaveAxis.McCamOut.ErrorID), '');
ELSIF NOT CamSlaveAxis.McCamOut.Error AND CamSlaveAxisAlarms[E_CamSlaveAxis.McCamOutError].bRaised THEN
	CamSlaveAxisAlarms[E_CamSlaveAxis.McCamOutError].Clear(0, 0);
END_IF

// ErrorID 4 - MC_CamTableSelect
IF CamSlaveAxis.MCCamTableSelect.Error AND NOT CamSlaveAxisAlarms[E_CamSlaveAxis.McLoadCamTableError].bRaised THEN
	RaiseAlarmWithStrings(Alarm := CamSlaveAxisAlarms[E_CamSlaveAxis.McLoadCamTableError], UDINT_TO_STRING(CamSlaveAxis.MCCamTableSelect.ErrorID), '');
ELSIF NOT CamSlaveAxis.MCCamTableSelect.Error AND CamSlaveAxisAlarms[E_CamSlaveAxis.McLoadCamTableError].bRaised THEN
	CamSlaveAxisAlarms[E_CamSlaveAxis.McLoadCamTableError].Clear(0, 0);
END_IF

// ErrorID 5 - MC_ReadCamTableSlaveDynamics
IF CamSlaveAxis.MCReadCamTableSlaveDynamics.Error AND NOT CamSlaveAxisAlarms[E_CamSlaveAxis.McReadSlaveDynamicsError].bRaised THEN
	RaiseAlarmWithStrings(Alarm := CamSlaveAxisAlarms[E_CamSlaveAxis.McReadSlaveDynamicsError], UDINT_TO_STRING(CamSlaveAxis.MCReadCamTableSlaveDynamics.ErrorID), '');
ELSIF NOT CamSlaveAxis.MCReadCamTableSlaveDynamics.Error AND CamSlaveAxisAlarms[E_CamSlaveAxis.McReadSlaveDynamicsError].bRaised THEN
	CamSlaveAxisAlarms[E_CamSlaveAxis.McReadSlaveDynamicsError].Clear(0, 0);
END_IF

// ErrorID 6 - MC_SetCamOnlineChangeMode 
IF CamSlaveAxis.MCSetCamOnlineChangeMode.Error AND NOT CamSlaveAxisAlarms[E_CamSlaveAxis.McCamOnlineChangeModeError].bRaised THEN
	RaiseAlarmWithStrings(Alarm := CamSlaveAxisAlarms[E_CamSlaveAxis.McCamOnlineChangeModeError], UDINT_TO_STRING(CamSlaveAxis.MCSetCamOnlineChangeMode.ErrorID), '');
ELSIF NOT CamSlaveAxis.MCSetCamOnlineChangeMode.Error AND CamSlaveAxisAlarms[E_CamSlaveAxis.McCamOnlineChangeModeError].bRaised THEN
	CamSlaveAxisAlarms[E_CamSlaveAxis.McCamOnlineChangeModeError].Clear(0, 0);
END_IF

// ErrorID 7 - MC_WriteMotionFunction
IF CamSlaveAxis.McWriteMotionFunction.Error AND NOT CamSlaveAxisAlarms[E_CamSlaveAxis.McWriteMotionFunctionError].bRaised THEN
	RaiseAlarmWithStrings(Alarm := CamSlaveAxisAlarms[E_CamSlaveAxis.McWriteMotionFunctionError], UDINT_TO_STRING(CamSlaveAxis.McWriteMotionFunction.ErrorID), '');
ELSIF NOT CamSlaveAxis.McWriteMotionFunction.Error AND CamSlaveAxisAlarms[E_CamSlaveAxis.McWriteMotionFunctionError].bRaised THEN
	CamSlaveAxisAlarms[E_CamSlaveAxis.McWriteMotionFunctionError].Clear(0, 0);
END_IF

// ErrorID 8 - MC_ReadParameterSet

// ErrorID 9 - CamControlSequenceError
IF CamSlaveAxis.SequenceError AND NOT CamSlaveAxisAlarms[E_CamSlaveAxis.CamControlSequenceError].bRaised THEN
	RaiseAlarmWithStrings(Alarm := CamSlaveAxisAlarms[E_CamSlaveAxis.CamControlSequenceError], UDINT_TO_STRING(CamSlaveAxis.SequenceErrorID), '');
ELSIF NOT CamSlaveAxis.SequenceError AND CamSlaveAxisAlarms[E_CamSlaveAxis.CamControlSequenceError].bRaised THEN
	CamSlaveAxisAlarms[E_CamSlaveAxis.CamControlSequenceError].Clear(0, 0);
END_IF

_CurrentAlarmSeverity := F_GetMaxSeverityRaised(Alarms := BasicAxisAlarms, CurrentSeverity := CurrentAlarmSeverity);
_CurrentAlarmSeverity := F_GetMaxSeverityRaised(Alarms := CamSlaveAxisAlarms, CurrentSeverity := CurrentAlarmSeverity);
END_METHOD

METHOD CyclicLogic
SUPER^.CyclicLogic();
CamSlaveAxis.CyclicLogic();
_Busy	 := CamSlaveAxis.Busy;
_Error	 := CamSlaveAxis.Error;
_ErrorID := CamSlaveAxis.ErrorID;
END_METHOD

// Basic component initialization logic
METHOD PROTECTED Initialize : BOOL;

// This method is called by CyclicLogic() as required
IF NOT CamSlaveAxis.InitComplete THEN
	RETURN;
END_IF

Initialize := SUPER^.Initialize();
END_METHOD

END_FUNCTION_BLOCK

// Communications/Modbus-RTU/FB_Component_ModbusRTUMaster
{attribute 'no_explicit_call' := 'do not call this POU directly'}
FUNCTION_BLOCK FB_Component_ModbusRTUMaster EXTENDS FB_ComponentBase IMPLEMENTS I_ModbusProvider
VAR
	ModbusAlarms   : ARRAY[1..MAX_MODBUS_ALARMS] OF FB_TcAlarm;
	Modbus		   : ModbusRtuMasterV2_KL6x22B;
	AsyncRequests  : FB_ModbusAsyncQueue;
	SyncRequests   : FB_ModbusSyncQueue;
	CurrentRequest : ST_ModbusRequest;
	State		   : (IDLE,
		GETNEXTREQUEST,
		GETNEXTWRITE,
		PROCESSWRITE,
		GETNEXTREAD,
		PROCESSREAD);
	CurrentRequestID : ULINT;
	ReadInProgress	 : BOOL;
	WriteInProgress	 : BOOL;
	SimTimer_TON	 : TON;
END_VAR

VAR CONSTANT
	MAX_MODBUS_ALARMS : DINT := 26;
END_VAR

METHOD PROTECTED CreateEvents
F_CreateAllEventsInClass(Alarms		:= ModbusAlarms,
						 ClassSize	:= SIZEOF(TC_EVENTS.MODBUSAlarms),
						 pInitEvent := ADR(TC_EVENTS.MODBUSAlarms.InitReferenceEvent),
						 Prefix		:= _Name);

SUPER^.CreateEvents();
END_METHOD

// This method serves as the entry point for all underlying FB logic
METHOD PUBLIC CyclicLogic
// This method should be called cyclically by descendant function blocks by invoking SUPER^.CyclicLogic().  Alternatively, the contents of this method could be reimplemented entirely in which case a call to this method would not be necessary.
VAR_INST
	OperationIndex	 : UDINT;
	CurrentOperation : ST_ModbusOperation;
	i				 : UDINT;
END_VAR
IF NOT _InitComplete THEN
	_InitComplete := Initialize();
	RETURN;
END_IF

_Busy := Modbus.BUSY;
CASE State OF
	IDLE:
		// Wait for requests
		Modbus(Execute := FALSE);
		IF SyncRequests.Count > 0 OR AsyncRequests.Count > 0 THEN
			State := GETNEXTREQUEST;
		END_IF

	GETNEXTREQUEST:
		IF NOT Modbus.BUSY THEN
			IF AsyncRequests.Count = 0 AND SyncRequests.Count > 0 THEN
				// No async requests--process next sync request
				CurrentRequest := SyncRequests.NextRequest;
				OperationIndex := 0;
				State		   := GETNEXTWRITE;
			ELSIF AsyncRequests.Count > 0 THEN
				// Process next async request
				CurrentRequest := AsyncRequests.NextRequest;
				AsyncRequests.Dequeue();
				OperationIndex := 0;
				State		   := GETNEXTWRITE;
			ELSE
				// No requests registered--go idle
				State := IDLE;
			END_IF
		END_IF

	GETNEXTWRITE:
		OperationIndex	 := OperationIndex + 1;
		CurrentOperation := CurrentRequest.WriteOps[OperationIndex];
		IF CurrentOperation.StartAddress <> 0 AND CurrentOperation.EndAddress <> 0 AND CurrentOperation.pAddress <> 0 THEN
			State := PROCESSWRITE;
		ELSE
			OperationIndex := 0;
			State		   := GETNEXTREAD;
		END_IF

	PROCESSWRITE:
		IF ProcessWrite(CurrentRequest.ipRequestor.SlaveID, CurrentOperation) THEN
			State := GETNEXTWRITE;
		END_IF

	GETNEXTREAD:
		OperationIndex	 := OperationIndex + 1;
		CurrentOperation := CurrentRequest.ReadOps[OperationIndex];
		IF CurrentOperation.StartAddress <> 0 AND CurrentOperation.EndAddress <> 0 AND CurrentOperation.pAddress <> 0 THEN
			State := PROCESSREAD;
		ELSE
			IF CurrentRequest.ipRequestor <> 0 THEN
				CurrentRequest.ipRequestor.ModbusRequestComplete(CurrentRequest.RequestID);
			END_IF

			State := GETNEXTREQUEST;
		END_IF

	PROCESSREAD:
		IF ProcessRead(CurrentRequest.ipRequestor.SlaveID, CurrentOperation) THEN
			State := GETNEXTREAD;
		END_IF
END_CASE

SUPER^.CyclicLogic();
_Busy := Modbus.BUSY;
END_METHOD

METHOD PROTECTED Initialize : BOOL;
Modbus.Timeout := Parameters_ModbusRTU.MODBUS_TIMEOUT;
Initialize	   := SUPER^.Initialize();
END_METHOD

METHOD PROTECTED Monitoring
IF Modbus.Error THEN
	CASE Modbus.ErrorId OF
		MODBUSERROR_ILLEGAL_FUNCTION:
			IF NOT ModbusAlarms[E_MODBUSAlarms.IllegalFunction].bRaised THEN
				ModbusAlarms[E_MODBUSAlarms.IllegalFunction].Raise(0);
			END_IF

		MODBUSERROR_ILLEGAL_DATA_ADDRESS:
			IF NOT ModbusAlarms[E_MODBUSAlarms.IllegalDataAddress].bRaised THEN
				ModbusAlarms[E_MODBUSAlarms.IllegalDataAddress].Raise(0);
			END_IF

		MODBUSERROR_ILLEGAL_DATA_VALUE:
			IF NOT ModbusAlarms[E_MODBUSAlarms.IllegalDataValue].bRaised THEN
				ModbusAlarms[E_MODBUSAlarms.IllegalDataValue].Raise(0);
			END_IF

		MODBUSERROR_SLAVE_DEVICE_FAILURE:
			IF NOT ModbusAlarms[E_MODBUSAlarms.SlaveDeviceFailure].bRaised THEN
				ModbusAlarms[E_MODBUSAlarms.SlaveDeviceFailure].Raise(0);
			END_IF

		MODBUSERROR_ACKNOWLEDGE:
			IF NOT ModbusAlarms[E_MODBUSAlarms.Acknowledge].bRaised THEN
				ModbusAlarms[E_MODBUSAlarms.Acknowledge].Raise(0);
			END_IF

		MODBUSERROR_SLAVE_DEVICE_BUSY:
			IF NOT ModbusAlarms[E_MODBUSAlarms.SlaveDeviceBusy].bRaised THEN
				ModbusAlarms[E_MODBUSAlarms.SlaveDeviceBusy].Raise(0);
			END_IF

		MODBUSERROR_NEGATIVE_ACKNOWLEDGE:
			IF NOT ModbusAlarms[E_MODBUSAlarms.NegativeAcknowledge].bRaised THEN
				ModbusAlarms[E_MODBUSAlarms.NegativeAcknowledge].Raise(0);
			END_IF

		MODBUSERROR_MEMORY_PARITY:
			IF NOT ModbusAlarms[E_MODBUSAlarms.MemoryParity].bRaised THEN
				ModbusAlarms[E_MODBUSAlarms.MemoryParity].Raise(0);
			END_IF

		MODBUSERROR_GATEWAY_PATH_UNAVAILABLE:
			IF NOT ModbusAlarms[E_MODBUSAlarms.GatewayPathUnavailable].bRaised THEN
				ModbusAlarms[E_MODBUSAlarms.GatewayPathUnavailable].Raise(0);
			END_IF

		MODBUSERROR_GATEWAY_TARGET_DEVICE_FAILED_TO_RESPOND:
			IF NOT ModbusAlarms[E_MODBUSAlarms.GatewayTargetDeviceFailedToRespond].bRaised THEN
				ModbusAlarms[E_MODBUSAlarms.GatewayTargetDeviceFailedToRespond].Raise(0);
			END_IF

		MODBUSERROR_CHARREC_TIMEOUT:
			IF NOT ModbusAlarms[E_MODBUSAlarms.CharRecTimeout].bRaised THEN
				ModbusAlarms[E_MODBUSAlarms.CharRecTimeout].Raise(0);
			END_IF

		MODBUSERROR_ILLEGAL_DATA_SIZE:
			IF NOT ModbusAlarms[E_MODBUSAlarms.IllegalDataSize].bRaised THEN
				ModbusAlarms[E_MODBUSAlarms.IllegalFunction].Raise(0);
			END_IF

		MODBUSERROR_ILLEGAL_DEVICE_ADDRESS:
			IF NOT ModbusAlarms[E_MODBUSAlarms.IllegalDataSize].bRaised THEN
				ModbusAlarms[E_MODBUSAlarms.IllegalFunction].Raise(0);
			END_IF

		MODBUSERROR_ILLEGAL_DESTINATION_ADDRESS:
			IF NOT ModbusAlarms[E_MODBUSAlarms.IllegalDestinationAddress].bRaised THEN
				ModbusAlarms[E_MODBUSAlarms.IllegalDestinationAddress].Raise(0);
			END_IF

		MODBUSERROR_ILLEGAL_DESTINATION_SIZE:
			IF NOT ModbusAlarms[E_MODBUSAlarms.IllegalDestinationSize].bRaised THEN
				ModbusAlarms[E_MODBUSAlarms.IllegalDestinationSize].Raise(0);
			END_IF

		MODBUSERROR_NO_RESPONSE:
			IF NOT ModbusAlarms[E_MODBUSAlarms.NoReponse].bRaised THEN
				ModbusAlarms[E_MODBUSAlarms.NoReponse].Raise(0);
			END_IF

		MODBUSERROR_TXBUFFOVERRUN:
			IF NOT ModbusAlarms[E_MODBUSAlarms.TxBufferOverrun].bRaised THEN
				ModbusAlarms[E_MODBUSAlarms.TxBufferOverrun].Raise(0);
			END_IF

		MODBUSERROR_SENDTIMEOUT:
			IF NOT ModbusAlarms[E_MODBUSAlarms.SendTimeout].bRaised THEN
				ModbusAlarms[E_MODBUSAlarms.SendTimeout].Raise(0);
			END_IF

		MODBUSERROR_DATASIZEOVERRUN:
			IF NOT ModbusAlarms[E_MODBUSAlarms.DataSizeOverrun].bRaised THEN
				ModbusAlarms[E_MODBUSAlarms.DataSizeOverrun].Raise(0);
			END_IF

		MODBUSERROR_STRINGOVERRUN:
			IF NOT ModbusAlarms[E_MODBUSAlarms.StringOverrun].bRaised THEN
				ModbusAlarms[E_MODBUSAlarms.StringOverrun].Raise(0);
			END_IF

		MODBUSERROR_INVALIDPOINTER:
			IF NOT ModbusAlarms[E_MODBUSAlarms.InvalidPointer].bRaised THEN
				ModbusAlarms[E_MODBUSAlarms.InvalidPointer].Raise(0);
			END_IF

		MODBUSERROR_CRC:
			IF NOT ModbusAlarms[E_MODBUSAlarms.CRCError].bRaised THEN
				ModbusAlarms[E_MODBUSAlarms.CRCError].Raise(0);
			END_IF

		MODBUSERROR_INVALIDMEMORYADDRESS:
			IF NOT ModbusAlarms[E_MODBUSAlarms.InvalidMemoryAddress].bRaised THEN
				ModbusAlarms[E_MODBUSAlarms.InvalidMemoryAddress].Raise(0);
			END_IF

		MODBUSERROR_TRANSMITBUFFERTOOSMALL:
			IF NOT ModbusAlarms[E_MODBUSAlarms.TransmitBufferTooSmall].bRaised THEN
				ModbusAlarms[E_MODBUSAlarms.TransmitBufferTooSmall].Raise(0);
			END_IF

	ELSE
		IF NOT ModbusAlarms[E_MODBUSAlarms.UnspecifiedError].bRaised THEN
			ModbusAlarms[E_MODBUSAlarms.UnspecifiedError].Raise(0);
		END_IF
	END_CASE
ELSE
	F_ClearAllEventsInClass(ModbusAlarms);
END_IF

SUPER^.Monitoring();
_CurrentAlarmSeverity := TcEventSeverity.Verbose;
_CurrentAlarmSeverity := F_GetMaxSeverityRaised(Alarms := ModbusAlarms, CurrentSeverity := _CurrentAlarmSeverity);
_Error				  := _CurrentAlarmSeverity >= TcEventSeverity.Error;
_ErrorID			  := TO_UDINT(Modbus.ErrorId);
END_METHOD

METHOD PUBLIC Reset : BOOL
Modbus(Execute := FALSE);
F_ClearAllEventsInClass(ModbusAlarms);
Reset := SUPER^.Reset();
END_METHOD

METHOD RegisterAsyncRequest : BOOL
VAR_INPUT
	Request : ST_ModbusRequest;
END_VAR

VAR_OUTPUT
	RequestID : ULINT;
END_VAR
IF Request.ipRequestor <> 0 THEN
	CurrentRequestID  := CurrentRequestID + 1;
	Request.RequestID := CurrentRequestID;
	IF AsyncRequests.Enqueue(Request) THEN
		RequestID			 := Request.RequestID;
		RegisterAsyncRequest := TRUE;
	END_IF
END_IF
END_METHOD

METHOD RegisterSyncRequest : BOOL
VAR_INPUT
	Request : ST_ModbusRequest;
END_VAR

VAR_OUTPUT
	RequestID : ULINT;
END_VAR
IF Request.ipRequestor <> 0 THEN
	CurrentRequestID  := CurrentRequestID + 1;
	Request.RequestID := CurrentRequestID;
	IF SyncRequests.Enqueue(Request) THEN
		RequestID			:= Request.RequestID;
		RegisterSyncRequest := TRUE;
	END_IF
END_IF
END_METHOD

METHOD ProcessRead : BOOL;
VAR_INPUT
	SlaveID	  : BYTE;
	Operation : ST_ModbusOperation;
END_VAR
IF _Simulate THEN
	SimTimer_TON(IN := TRUE, PT := T#100MS);
	IF SimTimer_TON.Q THEN
		SimTimer_TON(IN := FALSE);
		ProcessRead := TRUE;
	END_IF
ELSE
	IF ReadInProgress AND NOT Modbus.Busy THEN
		// Read complete
		Modbus.ReadRegs(UnitID		:= SlaveID,
						Quantity	:= (Operation.EndAddress - Operation.StartAddress),
						MBAddr		:= Operation.StartAddress,
						cbLength	:= (Operation.EndAddress - Operation.StartAddress) * 2,
						pMemoryAddr := Operation.pAddress,
						Timeout		:= Parameters_ModbusRTU.MODBUS_TIMEOUT,
						Execute		:= FALSE);

		ReadInProgress := FALSE;
		ProcessRead	   := TRUE;
	ELSE
		// Start read process
		Modbus.ReadRegs(UnitID		:= SlaveID,
						Quantity	:= (Operation.EndAddress - Operation.StartAddress),
						MBAddr		:= Operation.StartAddress,
						cbLength	:= (Operation.EndAddress - Operation.StartAddress) * 2,
						pMemoryAddr := Operation.pAddress,
						Timeout		:= Parameters_ModbusRTU.MODBUS_TIMEOUT,
						Execute		:= TRUE);

		IF Modbus.BUSY THEN
			ReadInProgress := TRUE;
		END_IF
	END_IF
END_IF
END_METHOD

METHOD ProcessWrite : BOOL;
VAR_INPUT
	SlaveID	  : BYTE;
	Operation : ST_ModbusOperation;
END_VAR
IF _Simulate THEN
	SimTimer_TON(IN := TRUE, PT := T#100MS);
	IF SimTimer_TON.Q THEN
		SimTimer_TON(IN := FALSE);
		ProcessWrite := TRUE;
	END_IF
ELSE
	IF WriteInProgress AND NOT Modbus.Busy THEN
		// Write complete
		Modbus.WriteRegs(UnitID		 := SlaveID,
						 Quantity	 := Operation.EndAddress - Operation.StartAddress,
						 MBAddr		 := Operation.StartAddress,
						 cbLength	 := (Operation.EndAddress - Operation.StartAddress) * 2,
						 pMemoryAddr := Operation.pAddress,
						 Timeout	 := Parameters_ModbusRTU.MODBUS_TIMEOUT,
						 Execute	 := FALSE);

		WriteInProgress := FALSE;
		ProcessWrite	:= TRUE;
	ELSE
		Modbus.WriteRegs(UnitID		 := SlaveID,
						 Quantity	 := Operation.EndAddress - Operation.StartAddress,
						 MBAddr		 := Operation.StartAddress,
						 cbLength	 := (Operation.EndAddress - Operation.StartAddress) * 2,
						 pMemoryAddr := Operation.pAddress,
						 Timeout	 := Parameters_ModbusRTU.MODBUS_TIMEOUT,
						 Execute	 := TRUE);

		IF Modbus.BUSY THEN
			WriteInProgress := TRUE;
		END_IF
	END_IF
END_IF
END_METHOD

END_FUNCTION_BLOCK

// Communications/Modbus-RTU/I_ModbusProvider
INTERFACE I_ModbusProvider

METHOD RegisterAsyncRequest : BOOL
VAR_INPUT
	Request : ST_ModbusRequest;
END_VAR

VAR_OUTPUT
	RequestID : ULINT;
END_VAR
END_METHOD

METHOD RegisterSyncRequest : BOOL
VAR_INPUT
	Request : ST_ModbusRequest;
END_VAR

VAR_OUTPUT
	RequestID : ULINT;
END_VAR
END_METHOD

END_INTERFACE

// Communications/Modbus-RTU/FB_ModbusAsyncQueue
{attribute 'no_explicit_call' := 'do not call this POU directly'}
{attribute 'hide'}
FUNCTION_BLOCK FB_ModbusAsyncQueue
VAR
	RequestsInQueue : UDINT := 0;
	Requests		: ARRAY[1..Parameters_ModbusRTU.MAX_MODBUS_REQUESTS] OF ST_ModbusRequest;
END_VAR

//	Method Clear() Brute force reset of buffer
METHOD Clear : BOOL
MEMSET(ADR(Requests), 0, SIZEOF(Requests));
RequestsInQueue := 0;
Clear			:= TRUE;
END_METHOD

PROPERTY Count : UDINT
GET
VAR
	i	 : UDINT;
	temp : UDINT;
END_VAR
Count := RequestsInQueue;
END_GET
END_PROPERTY

METHOD Dequeue : BOOL
IF RequestsInQueue > 0 THEN
	MEMSET(ADR(Requests[1]), 0, SIZEOF(Requests[1]));
	RequestsInQueue := RequestsInQueue - 1;
	IF RequestsInQueue > 0 THEN
		MEMMOVE(ADR(Requests[1]), ADR(Requests[2]), SIZEOF(Requests[2]) * RequestsInQueue);
		MEMSET(ADR(Requests[RequestsInQueue + 1]), 0, (SIZEOF(Requests[1]) * (Parameters_ModbusRTU.MAX_MODBUS_REQUESTS - RequestsInQueue)));
	END_IF

	Dequeue := TRUE;
END_IF
END_METHOD

METHOD Enqueue : BOOL
VAR_INPUT
	Request : ST_ModbusRequest;
END_VAR

VAR
	i : UDINT;
END_VAR
FOR i := 1 TO RequestsInQueue DO
	IF MEMCMP(ADR(Request), ADR(Requests[i]), SIZEOF(ST_ModbusRequest)) = 0 THEN
		Enqueue := TRUE;
		RETURN;
	END_IF
END_FOR

IF RequestsInQueue < Parameters_ModbusRTU.MAX_MODBUS_REQUESTS THEN
	RequestsInQueue			  := RequestsInQueue + 1;
	Requests[RequestsInQueue] := Request;
	Enqueue					  := TRUE;
END_IF
END_METHOD

PROPERTY NextRequest : ST_ModbusRequest
GET
IF RequestsInQueue > 0 THEN
	NextRequest := Requests[1];
END_IF
END_GET
END_PROPERTY

END_FUNCTION_BLOCK

// Communications/Modbus-RTU/FB_ModbusSyncQueue
{attribute 'no_explicit_call' := 'do not call this POU directly'}
{attribute 'hide'}
FUNCTION_BLOCK FB_ModbusSyncQueue
VAR
	RequestsInQueue : UDINT := 0;
	Requests		: ARRAY[1..Parameters_ModbusRTU.MAX_MODBUS_REQUESTS] OF ST_ModbusRequest;
	CurrentRequest	: UDINT;
END_VAR

//	Method Clear() Brute force reset of buffer
METHOD Clear : BOOL
MEMSET(ADR(Requests), 0, SIZEOF(Requests));
RequestsInQueue := 0;
Clear			:= TRUE;
END_METHOD

PROPERTY Count : UDINT
GET
VAR
	i	 : UDINT;
	temp : UDINT;
END_VAR
Count := RequestsInQueue;
END_GET
END_PROPERTY

METHOD Enqueue : BOOL
VAR_INPUT
	Request : ST_ModbusRequest;
END_VAR

VAR
	i : UDINT;
END_VAR
FOR i := 1 TO RequestsInQueue DO
	IF MEMCMP(ADR(Request), ADR(Requests[i]), SIZEOF(ST_ModbusRequest)) = 0 THEN
		Enqueue := TRUE;
		RETURN;
	END_IF
END_FOR

IF RequestsInQueue < Parameters_ModbusRTU.MAX_MODBUS_REQUESTS THEN
	RequestsInQueue			  := RequestsInQueue + 1;
	Requests[RequestsInQueue] := Request;
	Enqueue					  := TRUE;
END_IF
END_METHOD

PROPERTY NextRequest : ST_ModbusRequest
GET
IF RequestsInQueue > 0 THEN
	CurrentRequest := CurrentRequest + 1;
	IF CurrentRequest > RequestsInQueue THEN
		CurrentRequest := 1;
	END_IF

	NextRequest := Requests[CurrentRequest];
END_IF
END_GET
END_PROPERTY

END_FUNCTION_BLOCK

// Communications/Modbus-RTU/I_ModbusConsumer
INTERFACE I_ModbusConsumer

METHOD ModbusRequestComplete
VAR_INPUT
	RequestID : ULINT;
END_VAR
END_METHOD

PROPERTY SlaveID : BYTE
GET
END_GET
END_PROPERTY

END_INTERFACE

// PackML/FB_Component_PackML_EventHandler
FUNCTION_BLOCK FB_Component_PackML_EventHandler EXTENDS FB_ListenerBase2 IMPLEMENTS I_ComponentBase
VAR
	(* Base Component variables and Properties here **********************************************)

	// Base Component Properties
	_Error					   : BOOL;
	_ErrorID				   : UDINT;
	_InitComplete			   : BOOL;
	_InSimulation			   : BOOL;
	_Name					   : STRING;
	_ParentResponseDefinitions : ARRAY[0..4] OF SPT_BaseTypes.E_AlarmResponse;
	_Busy					   : BOOL;
	_CurrentAlarmSeverity	   : SPT_BaseTypes.TcEventSeverity;

	// Base Component HMI
	HMI : ST_ComponentBase_HMI;

	// Alarms
	PackMLEventHandlerAlarms : ARRAY[1..1] OF FB_TcAlarm;

	(* Event Handling Data starts here*******************************************************************)

	// Properties
	_AdminTag		  : REFERENCE TO Tc3_PackML_V2.ST_PMLa; // Reference to PML Admin Structure
	_InternalErrorAck : BOOL;								// Acknowledgement of internal Error
	_InternalError	  : BOOL;								// a internal Error is pending

	// Parameter Properties
	_AlarmToStopReason	 : BOOL; // Add Alarms to StopReason
	_WarningToStopReason : BOOL; // Add Warnings to Stopreason                                                              				

	// Count of Alarms
	CntAlarmsRaised : INT; // raised and not logged Alarm

	// Event Informations
	NewEvent		 : BOOL;											  // Event raised
	aEventInfoBuffer : ARRAY[1..Tc3_PackML_V2.MaxAlarms] OF ST_EventInfo; // incoming Event Info Buffer
	stEventInfo		 : ST_EventInfo;									  // temp Event Info Sructure

	// Alarm Array Counter
	UnclearedWarnings	 : DINT; // number of uncleared warnings
	UnclearedAlarms		 : DINT; // number of uncleared alarms
	UnclearedStopReasons : DINT; // number of uncleared stop reasons
	MsgInHistory		 : DINT; // number of messages in history

	// TimeZone
	fbTimeZone			: Tc2_Utilities.FB_GetTimeZoneInformation;			// Timezone information
	fbSpecificLocalTime : Tc2_Utilities.FB_SystemTimeToTzSpecificLocalTime; // Local time 
	GetTimeZone			: BOOL := TRUE;										// get timezone

	// Listener
	fbListenerFilter : FB_TcEventFilter; // instance of listener filter
	EventsSubscribed : BOOL;			 // Events subscibed
END_VAR

VAR CONSTANT
	cMsgCtrlMask : DWORD  := Tc2_System.ADSLOG_MSGTYPE_ERROR OR Tc2_System.ADSLOG_MSGTYPE_MSGBOX; // Internal Message TraceLevel
	cBaseMsg	 : STRING := 'FB_PackML_EventHandler Msg.: ';									  // base information for internal error message
END_VAR

PROPERTY AdminTag : REFERENCE TO Tc3_PackML_V2.ST_PMLa
SET
_AdminTag REF= AdminTag;
END_SET
END_PROPERTY

METHOD PRIVATE AlarmArrayHandler : HRESULT
VAR_INPUT
	pAlarmArray			 : POINTER TO ST_Alarm;	  // Pointer to Array of ST_Alarm of Alarm / Warning / Stop reason
	NewAlarm_Ref		 : REFERENCE TO ST_Alarm; // Reference to ST_Alarm of an new Alarm / Warning / Stop reason
	ActAlarmsCounter_Ref : REFERENCE TO DINT;	  // Reference to couter of active Alarm / Warning / Stop reason
	MaxArrayElements	 : INT;					  // max. Alarm / Warning / Stop reason constant
	BufferOverflow_Ref	 : REFERENCE TO BOOL;	  // Reference to BOOL Variable for Buffer Overflow information
END_VAR

VAR
	_Iterator				  : DINT; // FOR-Loop iterator						
	_MaxArrayElementsInternal : INT;  // calculated internal Array upper border
	_FiFo					  : BOOL; // Activate first in / first out function
END_VAR
IF __ISVALIDREF(NewAlarm_Ref) AND __ISVALIDREF(ActAlarmsCounter_Ref) AND __ISVALIDREF(BufferOverflow_Ref) AND pAlarmArray <> 0 THEN
	_MaxArrayElementsInternal := (MaxArrayElements - 1);

	// Move array down 1
	Tc2_System.MEMMOVE(destAddr := ADR(pAlarmArray[1]), srcAddr := ADR(pAlarmArray[0]), n := (SIZEOF(Tc3_PackML_V2.ST_Alarm) * TO_UINT(_MaxArrayElementsInternal))); // move Alarm 

	// Write new Alarm
	Tc2_System.MEMCPY(destAddr := ADR(pAlarmArray[0]), srcAddr := ADR(NewAlarm_Ref), n := SIZEOF(Tc3_PackML_V2.ST_Alarm)); // set Alarm 

	// Validate Alarm handled
	AlarmArrayHandler := S_OK;
ELSE
	// Set internal Error
	Tc2_System.ADSLOGSTR(msgCtrlMask := cMsgCtrlMask, msgFmtStr := Tc2_Standard.CONCAT(cBaseMsg, 'AlarmArrayHandler: %s'), strArg := 'Input-reference error');
	AlarmArrayHandler := E_FAIL;
	_InternalError	  := TRUE;
END_IF
END_METHOD

PROPERTY AlarmToStopReason : BOOL
SET
_AlarmToStopReason := AlarmToStopReason;
END_SET
END_PROPERTY

METHOD AllowHMIControl
HMI.Status.HMIControlAvailable := TRUE;
END_METHOD

METHOD BlockHMIControl
HMI.Status.HMIControlAvailable := FALSE;
END_METHOD

PROPERTY Busy : BOOL
GET
Busy := _Busy;
END_GET
END_PROPERTY

METHOD PRIVATE ClearStopReason : HRESULT
VAR_INPUT
	pAlarmArray		 : POINTER TO ST_Alarm; // Pointer to Array of ST_Alarm of Alarm / Warning / Stop reason
	ActAlarms_Ref	 : REFERENCE TO DINT;	// Reference to couter of active Alarm / Warning / Stop reason
	MaxArrayElements : INT;					// max. Alarm / Warning / Stop reason constant
	EventId			 : UDINT;				// EventId of Alarm / Warning / Stop reason to confirm
END_VAR

VAR
	_Iterator				  : INT;	 // FOR-Loop iterator	
	_Iterator2				  : DINT;	 // FOR-Loop iterator	
	_hr						  : HRESULT; // hresult
	_MaxArrayElementsInternal : INT;	 // calculated internal Array upper border
END_VAR
IF __ISVALIDREF(ActAlarms_Ref) THEN
	_MaxArrayElementsInternal := (MaxArrayElements - 1);

	// Search Alarm in Array
	FOR _Iterator := 0 TO _MaxArrayElementsInternal DO
		IF (pAlarmArray[_Iterator].ID = TO_DINT(EventId)) THEN
			// Delete Alarm	
			Tc2_System.MEMSET(ADR(pAlarmArray[_Iterator]), 0, SIZEOF(Tc3_PackML_V2.ST_Alarm));

			// Close empty entry in source array
			Tc2_System.MEMMOVE(destAddr := ADR(pAlarmArray[_Iterator]), srcAddr := ADR(pAlarmArray[_Iterator + 1]), n := (SIZEOF(Tc3_PackML_V2.ST_Alarm) * (TO_UINT((_MaxArrayElementsInternal) - (_Iterator))))); // move Alarm 
			Tc2_System.MEMSET(destAddr := ADR(pAlarmArray[_MaxArrayElementsInternal]), fillByte := 0, n := SIZEOF(Tc3_PackML_V2.ST_Alarm));																		   // delete last entry

			// Find next empty entry index 
			FOR _Iterator2 := 0 TO (_MaxArrayElementsInternal) DO
				IF (pAlarmArray[_Iterator2].Message = '') OR (_Iterator2 = _MaxArrayElementsInternal) THEN
					IF _Iterator2 > 0 THEN
						ActAlarms_Ref := _Iterator2 - 1;
					ELSE
						ActAlarms_Ref := _Iterator2;
					END_IF

					EXIT;
				END_IF
			END_FOR

			EXIT;
		END_IF
	END_FOR

	ClearStopReason := S_OK;
ELSE
	// Set internal Error
	Tc2_System.ADSLOGSTR(msgCtrlMask := cMsgCtrlMask, msgFmtStr := Tc2_Standard.CONCAT(cBaseMsg, 'ClearStopReason: %s'), strArg := 'Input-reference error');
	ClearStopReason := E_FAIL;
	_InternalError	:= TRUE;
END_IF
END_METHOD

METHOD PRIVATE ConfirmAlarm : HRESULT
VAR_INPUT
	pAlarmArray		 : POINTER TO ST_Alarm; // Pointer to Array of ST_Alarm of Alarm / Warning / Stop reason
	ActAlarms_Ref	 : REFERENCE TO DINT;	// Reference to couter of active Alarm / Warning / Stop reason
	MaxArrayElements : INT;					// max. Alarm / Warning / Stop reason constant
	EventId			 : UDINT;				// EventId of Alarm / Warning / Stop reason to confirm
	Timestamp		 : ULINT;				// Event Timestamp
END_VAR

VAR
	_Iterator				  : INT;		// FOR-Loop iterator	
	_TempTimestruct			  : TIMESTRUCT; // TimeStruct for ACK Time
	_MaxArrayElementsInternal : INT;		// calculated internal Array upper border
END_VAR
IF __ISVALIDREF(ActAlarms_Ref) THEN
	_MaxArrayElementsInternal := (MaxArrayElements - 1);

	// Search Alarm in Array
	FOR _Iterator := 0 TO _MaxArrayElementsInternal DO
		IF (pAlarmArray[_Iterator].ID = TO_DINT(EventId)) THEN
			// TimeZone
			THIS^.fbSpecificLocalTime(in := Tc2_Utilities.FILETIME64_TO_SYSTEMTIME(Timestamp), tzInfo := fbTimeZone.tzInfo, out => _TempTimestruct);

			// Set ACK Timestamp	
			pAlarmArray[_Iterator].AckDateTime[0] := TO_DINT(_TempTimestruct.wYear);
			pAlarmArray[_Iterator].AckDateTime[1] := TO_DINT(_TempTimestruct.wMonth);
			pAlarmArray[_Iterator].AckDateTime[2] := TO_DINT(_TempTimestruct.wDay);
			pAlarmArray[_Iterator].AckDateTime[3] := TO_DINT(_TempTimestruct.wHour);
			pAlarmArray[_Iterator].AckDateTime[4] := TO_DINT(_TempTimestruct.wMinute);
			pAlarmArray[_Iterator].AckDateTime[5] := TO_DINT(_TempTimestruct.wSecond);
			pAlarmArray[_Iterator].AckDateTime[6] := TO_DINT(_TempTimestruct.wMilliseconds);
			pAlarmArray[_Iterator].Trigger		  := FALSE;
			EXIT;
		END_IF
	END_FOR

	ConfirmAlarm := S_OK;
ELSE
	// Set internal Error
	Tc2_System.ADSLOGSTR(msgCtrlMask := cMsgCtrlMask, msgFmtStr := Tc2_Standard.CONCAT(cBaseMsg, 'ConfirmAlarm: %s'), strArg := 'Input-reference error');
	ConfirmAlarm   := E_FAIL;
	_InternalError := TRUE;
END_IF
END_METHOD

PROPERTY CurrentAlarmSeverity : SPT_BaseTypes.TcEventSeverity
GET
CurrentAlarmSeverity := _CurrentAlarmSeverity;
END_GET
END_PROPERTY

METHOD CyclicLogic
IF NOT InitComplete THEN
	_InitComplete := Initialize();
	RETURN;
END_IF

Execute();
_Busy		  := EventsSubscribed;
_Error		  := FALSE;
_ErrorID	  := 0;
_InSimulation := FALSE; // Does not use simulation
END_METHOD

PROPERTY Error : BOOL
GET
Error := _Error;
END_GET
END_PROPERTY

PROPERTY ErrorID : UDINT
GET
ErrorID := _ErrorID;
END_GET
END_PROPERTY

METHOD PUBLIC EventListener : HRESULT
VAR_INPUT
	Subscribe : BOOL; // Subscibe Events
END_VAR

VAR_OUTPUT
	Subscribed : BOOL; // Events are subscribed
END_VAR

